C09504=6449,32951,-27517,288,-27969,-3249
C09505=6447,32929,-27544,288,-27961,-3248
C09506=6439,32909,-27568,289,-27953,-3245
C09507=6438,32887,-27595,290,-27945,-3245
C09508=6431,32867,-27619,291,-27937,-3242
C09509=6424,32847,-27644,292,-27930,-3239
C09510=6417,32826,-27669,293,-27922,-3237
C09511=6410,32806,-27694,294,-27914,-3234
C09512=6403,32785,-27719,295,-27907,-3231
C09513=6396,32765,-27743,296,-27899,-3228
C09514=6388,32745,-27768,298,-27891,-3226
C09515=6381,32724,-27793,299,-27884,-3223
C09516=6374,32704,-27818,300,-27876,-3220
C09517=6356,32692,-27833,302,-27871,-3213
C09518=6356,32692,-26433,302,-27871,-3213
C09519=5833,33315,-23080,374,-28099,-3008
C09520=5833,33315,-27080,374,-28099,-3008
C09521=5810,33311,-27085,378,-28097,-2999
C09522=5793,33299,-27099,380,-28093,-2992
C09523=5770,33296,-27104,384,-28091,-2983
C09524=5747,33292,-27108,387,-28090,-2974
C09525=5724,33289,-27112,390,-28088,-2965
C09526=5701,33286,-27117,393,-28087,-2956
C09527=5678,33282,-27121,397,-28085,-2947
C09528=5657,33289,-27113,400,-28087,-2939
C09529=5634,33286,-27117,403,-28086,-2930
C09530=5614,33292,-27109,406,-28088,-2922
C09531=5592,33293,-27109,409,-28088,-2914
C09532=5571,33295,-27106,412,-28089,-2906
C09533=5550,33298,-27103,415,-28090,-2897
C09534=5528,33299,-27102,418,-28090,-2889
C09535=5508,33305,-27094,421,-28092,-2881
C09536=5487,33309,-27090,424,-28093,-2873
C09537=5464,33309,-27091,427,-28093,-2864
C09538=5444,33315,-27083,430,-28095,-2856
C09539=5424,33322,-27075,433,-28097,-2848
C09540=5405,33333,-27061,435,-28101,-2841
C09541=5387,33345,-27047,438,-28106,-2834
C09542=5367,33353,-27038,441,-28108,-2826
C09543=5356,33370,-27017,442,-28115,-2821
C09544=5365,33371,-27016,441,-28115,-2825
C09545=5386,33365,-27023,438,-28113,-2833
C09546=5404,33351,-27039,435,-28108,-2840
C09547=5424,33345,-27046,433,-28106,-2848
C09548=5443,33334,-27060,430,-28102,-2856
C09549=5463,33328,-27068,427,-28100,-2864
C09550=5485,33327,-27068,424,-28100,-2872
C09551=5507,33324,-27071,421,-28099,-2880
C09552=5527,33318,-27079,418,-28097,-2888
C09553=5548,33316,-27081,415,-28096,-2897
C09554=5570,33314,-27083,412,-28096,-2905
C09555=5590,33308,-27091,409,-28094,-2913
C09556=5613,33311,-27086,406,-28095,-2922
C09557=5633,33305,-27094,403,-28093,-2930
C09558=5656,33308,-27090,400,-28095,-2939
C09559=5677,33301,-27098,397,-28092,-2947
C09560=5700,33305,-27094,394,-28094,-2956
C09561=5723,33308,-27089,390,-28095,-2965
C09562=5746,33311,-27085,387,-28097,-2974
C09563=5769,33315,-27081,384,-28098,-2982
C09564=5792,33318,-27076,380,-28100,-2991
C09565=5810,33329,-27063,378,-28104,-2999
C09566=5832,33334,-27056,375,-28106,-3007
C09567=5850,33346,-27042,372,-28111,-3014
C09568=5864,33364,-27020,370,-28118,-3019
C09569=5880,33379,-27002,367,-28124,-3026
C09570=5893,33394,-26983,366,-28129,-3031
C09571=5902,33413,-26960,364,-28137,-3034
C09572=5916,33431,-26938,362,-28144,-3040
C09573=5937,33427,-26943,359,-28142,-3048
C09574=5926,33410,-26964,361,-28136,-3043
C09575=5911,33392,-26986,363,-28129,-3038
C09576=5897,33374,-27008,365,-28122,-3033
C09577=5883,33356,-27030,367,-28115,-3027
C09578=5869,33339,-27051,369,-28108,-3021
C09579=5851,33327,-27065,372,-28104,-3015
C09580=5833,33315,-27080,374,-28099,-3008
C09581=5833,33315,-25680,374,-28099,-3008
C09582=5638,33727,-22582,400,-28251,-2930
C09583=5638,33727,-26582,400,-28251,-2930
C09584=5614,33723,-26586,404,-28250,-2921
C09585=5590,33720,-26591,407,-28248,-2911
C09586=5566,33716,-26595,410,-28246,-2902
C09587=5542,33713,-26600,414,-28245,-2893
C09588=5518,33709,-26604,417,-28243,-2883
C09589=5494,33706,-26609,421,-28242,-2874
C09590=5470,33702,-26613,424,-28240,-2865
C09591=5446,33699,-26618,427,-28238,-2855
C09592=5422,33695,-26622,431,-28237,-2846
C09593=5435,33707,-26608,429,-28241,-2851
C09594=5459,33710,-26604,426,-28243,-2860
C09595=5483,33714,-26599,422,-28244,-2870
C09596=5507,33717,-26595,419,-28246,-2879
C09597=5531,33721,-26590,415,-28248,-2888
C09598=5555,33724,-26586,412,-28249,-2898
C09599=5573,33736,-26571,409,-28254,-2905
C09600=5597,33740,-26566,406,-28256,-2914
C09601=5621,33743,-26562,402,-28257,-2924
C09602=5645,33747,-26557,399,-28259,-2933
C09603=5667,33754,-26549,396,-28262,-2941
C09604=5688,33763,-26538,393,-28265,-2949
C09605=5712,33766,-26533,389,-28267,-2959
C09606=5730,33779,-26518,387,-28272,-2966
C09607=5754,33782,-26514,383,-28273,-2975
C09608=5774,33792,-26502,380,-28277,-2983
C09609=5797,33798,-26494,377,-28280,-2992
C09610=5815,33810,-26479,374,-28284,-2999
C09611=5837,33817,-26471,371,-28287,-3008
C09612=5856,33830,-26455,369,-28292,-3015
C09613=5874,33842,-26440,366,-28297,-3022
C09614=5892,33855,-26424,363,-28302,-3029
C09615=5908,33872,-26404,361,-28308,-3035
C09616=5925,33886,-26386,358,-28314,-3042
C09617=5940,33905,-26363,356,-28321,-3047
C09618=5958,33917,-26348,354,-28326,-3055
C09619=5973,33936,-26325,352,-28333,-3060
C09620=5988,33955,-26302,349,-28340,-3066
C09621=6000,33974,-26279,347,-28348,-3071
C09622=6015,33978,-26273,345,-28350,-3076
C09623=6017,33959,-24896,345,-28342,-3077
C09624=-41004,59868,4099,4900,-34257,16705
C09625=-41004,59868,1099,4900,-34257,16705
C09626=-41004,64596,1380,5213,-31659,16463
C09627=-41004,59868,1099,4900,-34257,16705
C09628=-41004,59868,9099,4900,-34257,16705
C09629=6017,33959,-22296,345,-28342,-3077
C09630=6017,33959,-26296,345,-28342,-3077
C09631=6002,33941,-26319,347,-28335,-3072
C09632=5988,33922,-26342,349,-28328,-3066
C09633=5973,33903,-26365,352,-28321,-3060
C09634=5955,33891,-26380,354,-28316,-3053
C09635=5940,33872,-26403,356,-28309,-3048
C09636=5922,33859,-26419,359,-28304,-3041
C09637=5906,33843,-26439,361,-28298,-3034
C09638=5887,33830,-26454,364,-28293,-3027
C09639=5869,33818,-26469,367,-28288,-3020
C09640=5850,33806,-26484,370,-28283,-3013
C09641=5832,33793,-26499,372,-28278,-3006
C09642=5811,33784,-26511,375,-28274,-2998
C09643=5789,33778,-26519,378,-28272,-2989
C09644=5771,33765,-26534,381,-28267,-2982
C09645=5747,33762,-26538,384,-28265,-2972
C09646=5726,33752,-26550,387,-28262,-2965
C09647=5704,33746,-26558,391,-28259,-2956
C09648=5680,33743,-26562,394,-28257,-2947
C09649=5660,33733,-26573,397,-28254,-2939
C09650=5638,33727,-26582,400,-28251,-2930
C09651=5638,33727,-25182,400,-28251,-2930
C09652=5388,35827,-20036,425,-29034,-2826
C09653=5388,35827,-24036,425,-29034,-2826
C09654=5365,35833,-24029,428,-29036,-2816
C09655=5342,35839,-24021,431,-29038,-2807
C09656=5318,35845,-24014,434,-29040,-2798
C09657=5295,35851,-24007,438,-29042,-2789
C09658=5271,35857,-24000,441,-29044,-2780
C09659=5248,35863,-23993,444,-29046,-2770
C09660=5223,35866,-23990,448,-29047,-2761
C09661=5200,35874,-23980,451,-29050,-2752
C09662=5176,35876,-23979,454,-29050,-2742
C09663=5151,35878,-23976,457,-29050,-2732
C09664=5128,35884,-23969,461,-29052,-2723
C09665=5104,35887,-23965,464,-29053,-2714
C09666=5078,35886,-23967,468,-29052,-2704
C09667=5054,35890,-23962,471,-29054,-2694
C09668=5029,35888,-23965,474,-29053,-2684
C09669=5005,35893,-23959,478,-29054,-2675
C09670=4979,35891,-23963,481,-29053,-2665
C09671=4953,35887,-23968,485,-29051,-2655
C09672=4930,35893,-23960,488,-29053,-2645
C09673=4904,35889,-23965,492,-29051,-2635
C09674=4878,35885,-23970,495,-29049,-2625
C09675=4852,35881,-23975,499,-29047,-2615
C09676=4826,35877,-23980,503,-29046,-2604
C09677=4799,35874,-23985,506,-29044,-2594
C09678=4773,35870,-23990,510,-29042,-2584
C09679=4747,35866,-23995,513,-29040,-2574
C09680=4721,35862,-24000,517,-29038,-2564
C09681=4700,35849,-24016,520,-29033,-2555
C09682=4674,35845,-24021,524,-29032,-2545
C09683=4686,35862,-24001,522,-29038,-2550
C09684=4710,35870,-23991,519,-29041,-2559
C09685=4736,35874,-23986,515,-29043,-2569
C09686=4762,35878,-23981,511,-29045,-2579
C09687=4788,35881,-23976,508,-29047,-2590
C09688=4814,35885,-23971,504,-29048,-2600
C09689=4840,35889,-23966,500,-29050,-2610
C09690=4866,35893,-23961,497,-29052,-2620
C09691=4892,35897,-23956,493,-29054,-2631
C09692=4918,35901,-23951,490,-29056,-2641
C09693=4944,35905,-23946,486,-29057,-2651
C09694=4970,35908,-23941,482,-29059,-2661
C09695=4996,35912,-23936,479,-29061,-2671
C09696=5020,35906,-23943,476,-29059,-2681
C09697=5046,35910,-23938,472,-29061,-2691
C09698=5069,35904,-23945,469,-29059,-2700
C09699=5094,35903,-23946,465,-29059,-2710
C09700=5119,35902,-23948,462,-29059,-2720
C09701=5143,35900,-23950,458,-29058,-2729
C09702=5168,35898,-23951,455,-29058,-2739
C09703=5192,35893,-23957,452,-29057,-2748
C09704=5215,35887,-23964,449,-29055,-2757
C09705=5238,35881,-23971,445,-29053,-2767
C09706=5262,35875,-23978,442,-29051,-2776
C09707=5286,35870,-23985,439,-29049,-2785
C09708=5310,35868,-23986,435,-29049,-2795
C09709=5333,35860,-23996,432,-29046,-2804
C09710=5358,35858,-23998,429,-29046,-2814
C09711=5381,35849,-24008,426,-29043,-2823
C09712=5402,35834,-24027,423,-29037,-2831
C09713=5388,35827,-24036,425,-29034,-2826
C09714=5388,35827,-22636,425,-29034,-2826
C09715=5324,36018,-19804,433,-29105,-2800
C09716=5324,36018,-23804,433,-29105,-2800
C09717=5298,36029,-23791,436,-29109,-2790
C09718=5273,36040,-23779,440,-29112,-2780
C09719=5249,36057,-23757,443,-29119,-2770
C09720=5224,36068,-23745,446,-29122,-2760
C09721=5200,36085,-23724,450,-29129,-2751
C09722=5175,36096,-23711,453,-29132,-2741
C09723=5149,36107,-23699,457,-29136,-2731
C09724=5126,36123,-23679,460,-29142,-2721
C09725=5100,36135,-23665,463,-29146,-2712
C09726=5075,36144,-23654,467,-29149,-2701
C09727=5048,36150,-23647,470,-29151,-2691
C09728=5024,36166,-23629,474,-29156,-2681
C09729=4997,36171,-23622,477,-29158,-2671
C09730=4972,36181,-23611,481,-29161,-2661
C09731=4947,36191,-23598,484,-29165,-2651
C09732=4920,36198,-23590,488,-29167,-2640
C09733=4893,36204,-23584,491,-29169,-2630
C09734=4867,36209,-23577,495,-29170,-2620
C09735=4840,36215,-23571,499,-29172,-2609
C09736=4814,36223,-23561,502,-29175,-2599
C09737=4787,36227,-23557,506,-29176,-2588
C09738=4760,36232,-23551,510,-29177,-2578
C09739=4734,36237,-23545,513,-29179,-2567
C09740=4706,36238,-23545,517,-29179,-2556
C09741=4678,36239,-23544,521,-29179,-2545
C09742=4651,36244,-23537,524,-29180,-2535
C09743=4623,36241,-23541,528,-29179,-2523
C09744=4596,36246,-23536,532,-29180,-2513
C09745=4566,36241,-23542,536,-29178,-2501
C09746=4562,36258,-23522,537,-29184,-2500
C09747=4588,36254,-23526,533,-29183,-2510
C09748=4617,36258,-23521,529,-29185,-2521
C09749=4646,36263,-23515,525,-29187,-2533
C09750=4673,36257,-23522,521,-29185,-2543
C09751=4699,36252,-23528,518,-29184,-2554
C09752=4728,36255,-23524,514,-29185,-2565
C09753=4755,36250,-23529,510,-29184,-2575
C09754=4782,36245,-23535,507,-29182,-2586
C09755=4808,36239,-23542,503,-29181,-2596
C09756=4835,36233,-23549,499,-29179,-2607
C09757=4862,36230,-23553,496,-29178,-2618
C09758=4888,36222,-23562,492,-29175,-2628
C09759=4915,36216,-23568,488,-29174,-2638
C09760=4942,36211,-23575,485,-29172,-2649
C09761=4967,36201,-23586,481,-29169,-2659
C09762=4992,36191,-23598,478,-29165,-2669
C09763=5019,36184,-23606,474,-29163,-2679
C09764=5045,36177,-23615,471,-29161,-2690
C09765=5070,36163,-23631,467,-29156,-2699
C09766=5096,36155,-23640,464,-29153,-2710
C09767=5120,36141,-23657,460,-29149,-2719
C09768=5145,36127,-23674,457,-29143,-2729
C09769=5170,36116,-23686,454,-29140,-2739
C09770=5195,36106,-23699,450,-29136,-2749
C09771=5219,36089,-23719,447,-29130,-2758
C09772=5244,36078,-23733,444,-29126,-2768
C09773=5268,36060,-23754,440,-29120,-2778
C09774=5293,36049,-23766,437,-29116,-2788
C09775=5317,36032,-23788,434,-29110,-2797
C09776=5324,36018,-23804,433,-29105,-2800
C09777=5324,36018,-22404,433,-29105,-2800
C09778=5373,36428,-19306,424,-29259,-2818
C09779=5373,36428,-23306,424,-29259,-2818
C09780=5363,36436,-23296,426,-29262,-2814
C09781=5350,36436,-23296,427,-29262,-2809
C09782=5340,36444,-23287,429,-29265,-2805
C09783=5330,36452,-23277,430,-29268,-2801
C09784=5320,36460,-23268,431,-29271,-2797
C09785=5309,36467,-23259,433,-29273,-2793
C09786=5299,36475,-23250,434,-29276,-2789
C09787=5289,36483,-23240,436,-29279,-2785
C09788=5278,36491,-23231,437,-29282,-2780
C09789=5268,36498,-23222,438,-29284,-2776
C09790=5258,36506,-23213,440,-29287,-2772
C09791=5248,36514,-23203,441,-29290,-2768
C09792=5237,36521,-23194,442,-29293,-2764
C09793=5227,36529,-23185,444,-29295,-2760
C09794=5215,36530,-23184,446,-29295,-2755
C09795=5205,36538,-23175,447,-29298,-2751
C09796=5195,36545,-23166,448,-29301,-2747
C09797=5184,36553,-23156,450,-29304,-2743
C09798=5174,36561,-23147,451,-29306,-2739
C09799=5162,36561,-21746,453,-29306,-2734
C09800=-41004,59868,4099,4900,-34257,16705
C09801=-41004,59868,1099,4900,-34257,16705
C09802=-41004,64596,1380,5213,-31659,16463
C09803=-41004,59868,1099,4900,-34257,16705
C09804=-41004,59868,9099,4900,-34257,16705
C09805=5162,36561,-19146,453,-29306,-2734
C09806=5162,36561,-23146,453,-29306,-2734
C09807=5152,36569,-23137,454,-29309,-2730
C09808=5142,36577,-23128,455,-29312,-2726
C09809=5131,36584,-23120,457,-29314,-2722
C09810=5119,36585,-23118,458,-29315,-2718
C09811=5109,36593,-23109,460,-29317,-2713
C09812=5098,36598,-23103,461,-29319,-2709
C09813=5087,36601,-23099,463,-29320,-2705
C09814=5081,36612,-23086,464,-29324,-2702
C09815=5079,36624,-23072,464,-29329,-2702
C09816=5090,36616,-23081,462,-29326,-2706
C09817=5102,36615,-23082,461,-29326,-2711
C09818=5113,36610,-23088,459,-29324,-2715
C09819=5124,36607,-23092,458,-29323,-2719
C09820=5134,36599,-23101,456,-29320,-2723
C09821=5145,36592,-23110,455,-29317,-2727
C09822=5156,36588,-23115,453,-29316,-2732
C09823=5167,36583,-23120,452,-29315,-2736
C09824=5177,36575,-23129,451,-29312,-2740
C09825=5187,36568,-23139,449,-29309,-2744
C09826=5199,36565,-23141,448,-29308,-2749
C09827=5210,36559,-23148,446,-29306,-2753
C09828=5220,36552,-23158,445,-29304,-2757
C09829=5230,36544,-23167,443,-29301,-2761
C09830=5240,36536,-23176,442,-29298,-2765
C09831=5251,36528,-23186,441,-29295,-2769
C09832=5261,36521,-23195,439,-29293,-2773
C09833=5271,36513,-23204,438,-29290,-2778
C09834=5281,36505,-23213,437,-29287,-2782
C09835=5293,36502,-23216,435,-29286,-2786
C09836=5304,36497,-23223,433,-29284,-2790
C09837=5314,36489,-23232,432,-29281,-2794
C09838=5324,36481,-23242,431,-29279,-2799
C09839=5335,36474,-23251,429,-29276,-2803
C09840=5345,36466,-23260,428,-29273,-2807
C09841=5355,36458,-23269,427,-29271,-2811
C09842=5365,36450,-23279,425,-29268,-2815
C09843=5376,36443,-23288,424,-29265,-2819
C09844=5386,36435,-23297,422,-29262,-2823
C09845=5386,36430,-23303,423,-29260,-2823
C09846=5373,36428,-23306,424,-29259,-2818
C09847=5373,36428,-21906,424,-29259,-2818
//INST
///DATE 2026/04/29 10:00
///ATTR SC,RW
///GROUP1 RB1
NOP
MOVJ C00000 VJ=0.78
MOVJ C00001 VJ=0.78
MOVL C00002 V=11.7
TIMER T=2.00
MOVL C00003 V=11.7
MOVJ C00004 VJ=0.78
MOVJ C00005 VJ=0.78
MOVJ C00006 VJ=0.78
MOVL C00007 V=8.0
MOVL C00008 V=8.0
MOVL C00009 V=8.0
MOVL C00010 V=8.0
MOVL C00011 V=8.0
MOVL C00012 V=8.0
MOVL C00013 V=8.0
MOVL C00014 V=8.0
MOVL C00015 V=8.0
MOVL C00016 V=8.0
MOVL C00017 V=8.0
MOVL C00018 V=8.0
MOVL C00019 V=8.0
MOVL C00020 V=8.0
MOVL C00021 V=8.0
MOVL C00022 V=8.0
MOVL C00023 V=8.0
MOVL C00024 V=8.0
MOVL C00025 V=8.0
MOVL C00026 V=8.0
MOVL C00027 V=8.0
MOVL C00028 V=8.0
MOVL C00029 V=8.0
MOVL C00030 V=8.0
MOVL C00031 V=8.0
MOVL C00032 V=8.0
MOVL C00033 V=8.0
MOVL C00034 V=8.0
MOVL C00035 V=8.0
MOVL C00036 V=8.0
MOVL C00037 V=8.0
MOVL C00038 V=8.0
MOVL C00039 V=8.0
MOVL C00040 V=8.0
MOVL C00041 V=8.0
MOVL C00042 V=8.0
MOVL C00043 V=8.0
MOVL C00044 V=8.0
MOVL C00045 V=8.0
MOVL C00046 V=8.0
MOVL C00047 V=8.0
MOVL C00048 V=8.0
MOVL C00049 V=8.0
MOVL C00050 V=8.0
MOVL C00051 V=8.0
MOVL C00052 V=8.0
MOVL C00053 V=8.0
MOVL C00054 V=8.0
MOVL C00055 V=8.0
MOVL C00056 V=8.0
MOVL C00057 V=8.0
MOVL C00058 V=8.0
MOVL C00059 V=8.0
MOVL C00060 V=8.0
MOVL C00061 V=8.0
MOVL C00062 V=8.0
MOVL C00063 V=8.0
MOVL C00064 V=8.0
MOVL C00065 V=8.0
MOVL C00066 V=8.0
MOVL C00067 V=8.0
MOVL C00068 V=8.0
MOVJ C00069 VJ=0.78
MOVL C00070 V=8.0
MOVL C00071 V=8.0
MOVL C00072 V=8.0
MOVL C00073 V=8.0
MOVL C00074 V=8.0
MOVL C00075 V=8.0
MOVL C00076 V=8.0
MOVL C00077 V=8.0
MOVL C00078 V=8.0
MOVL C00079 V=8.0
MOVL C00080 V=8.0
MOVL C00081 V=8.0
MOVL C00082 V=8.0
MOVL C00083 V=8.0
MOVL C00084 V=8.0
MOVL C00085 V=8.0
MOVL C00086 V=8.0
MOVL C00087 V=8.0
MOVL C00088 V=8.0
MOVL C00089 V=8.0
MOVL C00090 V=8.0
MOVL C00091 V=8.0
MOVL C00092 V=8.0
MOVL C00093 V=8.0
MOVL C00094 V=8.0
MOVL C00095 V=8.0
MOVL C00096 V=8.0
MOVL C00097 V=8.0
MOVL C00098 V=8.0
MOVL C00099 V=8.0
MOVL C00100 V=8.0
MOVL C00101 V=8.0
MOVL C00102 V=8.0
MOVL C00103 V=8.0
MOVL C00104 V=8.0
MOVL C00105 V=8.0
MOVL C00106 V=8.0
MOVL C00107 V=8.0
MOVL C00108 V=8.0
MOVL C00109 V=8.0
MOVL C00110 V=8.0
MOVL C00111 V=8.0
MOVL C00112 V=8.0
MOVL C00113 V=8.0
MOVL C00114 V=8.0
MOVL C00115 V=8.0
MOVL C00116 V=8.0
MOVL C00117 V=8.0
MOVL C00118 V=8.0
MOVL C00119 V=8.0
MOVL C00120 V=8.0
MOVL C00121 V=8.0
MOVL C00122 V=8.0
MOVL C00123 V=8.0
MOVL C00124 V=8.0
MOVL C00125 V=8.0
MOVL C00126 V=8.0
MOVL C00127 V=8.0
MOVL C00128 V=8.0
MOVL C00129 V=8.0
MOVL C00130 V=8.0
MOVL C00131 V=8.0
MOVJ C00132 VJ=0.78
MOVL C00133 V=8.0
MOVL C00134 V=8.0
MOVL C00135 V=8.0
MOVL C00136 V=8.0
MOVL C00137 V=8.0
MOVL C00138 V=8.0
MOVL C00139 V=8.0
MOVL C00140 V=8.0
MOVL C00141 V=8.0
MOVL C00142 V=8.0
MOVL C00143 V=8.0
MOVL C00144 V=8.0
MOVL C00145 V=8.0
MOVL C00146 V=8.0
MOVL C00147 V=8.0
MOVL C00148 V=8.0
MOVL C00149 V=8.0
MOVL C00150 V=8.0
MOVL C00151 V=8.0
MOVL C00152 V=8.0
MOVL C00153 V=8.0
MOVL C00154 V=8.0
MOVL C00155 V=8.0
MOVL C00156 V=8.0
MOVL C00157 V=8.0
MOVL C00158 V=8.0
MOVL C00159 V=8.0
MOVL C00160 V=8.0
MOVL C00161 V=8.0
MOVL C00162 V=8.0
MOVL C00163 V=8.0
MOVL C00164 V=8.0
MOVL C00165 V=8.0
MOVL C00166 V=8.0
MOVL C00167 V=8.0
MOVL C00168 V=8.0
MOVL C00169 V=8.0
MOVL C00170 V=8.0
MOVL C00171 V=8.0
MOVL C00172 V=8.0
MOVL C00173 V=8.0
MOVJ C00174 VJ=0.78
MOVJ C00175 VJ=0.78
MOVL C00176 V=11.7
TIMER T=2.00
MOVL C00177 V=11.7
MOVJ C00178 VJ=0.78
MOVJ C00179 VJ=0.78
MOVL C00180 V=8.0
MOVL C00181 V=8.0
MOVL C00182 V=8.0
MOVL C00183 V=8.0
MOVL C00184 V=8.0
MOVL C00185 V=8.0
MOVL C00186 V=8.0
MOVL C00187 V=8.0
MOVL C00188 V=8.0
MOVL C00189 V=8.0
MOVL C00190 V=8.0
MOVL C00191 V=8.0
MOVL C00192 V=8.0
MOVL C00193 V=8.0
MOVL C00194 V=8.0
MOVL C00195 V=8.0
MOVL C00196 V=8.0
MOVL C00197 V=8.0
MOVL C00198 V=8.0
MOVL C00199 V=8.0
MOVL C00200 V=8.0
MOVL C00201 V=8.0
MOVJ C00202 VJ=0.78
MOVL C00203 V=8.0
MOVL C00204 V=8.0
MOVL C00205 V=8.0
MOVL C00206 V=8.0
MOVL C00207 V=8.0
MOVL C00208 V=8.0
MOVL C00209 V=8.0
MOVL C00210 V=8.0
MOVL C00211 V=8.0
MOVL C00212 V=8.0
MOVL C00213 V=8.0
MOVL C00214 V=8.0
MOVL C00215 V=8.0
MOVL C00216 V=8.0
MOVL C00217 V=8.0
MOVL C00218 V=8.0
MOVL C00219 V=8.0
MOVL C00220 V=8.0
MOVL C00221 V=8.0
MOVL C00222 V=8.0
MOVL C00223 V=8.0
MOVL C00224 V=8.0
MOVL C00225 V=8.0
MOVL C00226 V=8.0
MOVL C00227 V=8.0
MOVL C00228 V=8.0
MOVL C00229 V=8.0
MOVL C00230 V=8.0
MOVL C00231 V=8.0
MOVL C00232 V=8.0
MOVL C00233 V=8.0
MOVL C00234 V=8.0
MOVL C00235 V=8.0
MOVL C00236 V=8.0
MOVL C00237 V=8.0
MOVL C00238 V=8.0
MOVL C00239 V=8.0
MOVL C00240 V=8.0
MOVL C00241 V=8.0
MOVL C00242 V=8.0
MOVL C00243 V=8.0
MOVL C00244 V=8.0
MOVL C00245 V=8.0
MOVL C00246 V=8.0
MOVL C00247 V=8.0
MOVL C00248 V=8.0
MOVL C00249 V=8.0
MOVL C00250 V=8.0
MOVL C00251 V=8.0
MOVL C00252 V=8.0
MOVL C00253 V=8.0
MOVL C00254 V=8.0
MOVL C00255 V=8.0
MOVL C00256 V=8.0
MOVL C00257 V=8.0
MOVL C00258 V=8.0
MOVL C00259 V=8.0
MOVL C00260 V=8.0
MOVL C00261 V=8.0
MOVL C00262 V=8.0
MOVL C00263 V=8.0
MOVL C00264 V=8.0
MOVJ C00265 VJ=0.78
MOVL C00266 V=8.0
MOVL C00267 V=8.0
MOVL C00268 V=8.0
MOVL C00269 V=8.0
MOVL C00270 V=8.0
MOVL C00271 V=8.0
MOVL C00272 V=8.0
MOVL C00273 V=8.0
MOVL C00274 V=8.0
MOVL C00275 V=8.0
MOVL C00276 V=8.0
MOVL C00277 V=8.0
MOVL C00278 V=8.0
MOVL C00279 V=8.0
MOVL C00280 V=8.0
MOVL C00281 V=8.0
MOVL C00282 V=8.0
MOVL C00283 V=8.0
MOVL C00284 V=8.0
MOVL C00285 V=8.0
MOVL C00286 V=8.0
MOVL C00287 V=8.0
MOVL C00288 V=8.0
MOVL C00289 V=8.0
MOVL C00290 V=8.0
MOVL C00291 V=8.0
MOVL C00292 V=8.0
MOVL C00293 V=8.0
MOVL C00294 V=8.0
MOVL C00295 V=8.0
MOVL C00296 V=8.0
MOVL C00297 V=8.0
MOVL C00298 V=8.0
MOVL C00299 V=8.0
MOVL C00300 V=8.0
MOVL C00301 V=8.0
MOVL C00302 V=8.0
MOVL C00303 V=8.0
MOVL C00304 V=8.0
MOVL C00305 V=8.0
MOVL C00306 V=8.0
MOVL C00307 V=8.0
MOVL C00308 V=8.0
MOVL C00309 V=8.0
MOVL C00310 V=8.0
MOVL C00311 V=8.0
MOVL C00312 V=8.0
MOVL C00313 V=8.0
MOVL C00314 V=8.0
MOVL C00315 V=8.0
MOVL C00316 V=8.0
MOVL C00317 V=8.0
MOVL C00318 V=8.0
MOVL C00319 V=8.0
MOVL C00320 V=8.0
MOVL C00321 V=8.0
MOVL C00322 V=8.0
MOVL C00323 V=8.0
MOVL C00324 V=8.0
MOVL C00325 V=8.0
MOVL C00326 V=8.0
MOVL C00327 V=8.0
MOVJ C00328 VJ=0.78
MOVL C00329 V=8.0
MOVL C00330 V=8.0
MOVL C00331 V=8.0
MOVL C00332 V=8.0
MOVL C00333 V=8.0
MOVL C00334 V=8.0
MOVL C00335 V=8.0
MOVL C00336 V=8.0
MOVL C00337 V=8.0
MOVL C00338 V=8.0
MOVL C00339 V=8.0
MOVL C00340 V=8.0
MOVL C00341 V=8.0
MOVL C00342 V=8.0
MOVL C00343 V=8.0
MOVL C00344 V=8.0
MOVL C00345 V=8.0
MOVL C00346 V=8.0
MOVL C00347 V=8.0
MOVL C00348 V=8.0
MOVL C00349 V=8.0
MOVJ C00350 VJ=0.78
MOVJ C00351 VJ=0.78
MOVL C00352 V=11.7
TIMER T=2.00
MOVL C00353 V=11.7
MOVJ C00354 VJ=0.78
MOVJ C00355 VJ=0.78
MOVL C00356 V=8.0
MOVL C00357 V=8.0
MOVL C00358 V=8.0
MOVL C00359 V=8.0
MOVL C00360 V=8.0
MOVL C00361 V=8.0
MOVL C00362 V=8.0
MOVL C00363 V=8.0
MOVL C00364 V=8.0
MOVL C00365 V=8.0
MOVL C00366 V=8.0
MOVL C00367 V=8.0
MOVL C00368 V=8.0
MOVL C00369 V=8.0
MOVL C00370 V=8.0
MOVL C00371 V=8.0
MOVL C00372 V=8.0
MOVL C00373 V=8.0
MOVL C00374 V=8.0
MOVL C00375 V=8.0
MOVL C00376 V=8.0
MOVL C00377 V=8.0
MOVL C00378 V=8.0
MOVL C00379 V=8.0
MOVL C00380 V=8.0
MOVL C00381 V=8.0
MOVL C00382 V=8.0
MOVL C00383 V=8.0
MOVL C00384 V=8.0
MOVL C00385 V=8.0
MOVL C00386 V=8.0
MOVL C00387 V=8.0
MOVL C00388 V=8.0
MOVL C00389 V=8.0
MOVL C00390 V=8.0
MOVL C00391 V=8.0
MOVL C00392 V=8.0
MOVL C00393 V=8.0
MOVL C00394 V=8.0
MOVL C00395 V=8.0
MOVL C00396 V=8.0
MOVL C00397 V=8.0
MOVJ C00398 VJ=0.78
MOVL C00399 V=8.0
MOVL C00400 V=8.0
MOVL C00401 V=8.0
MOVL C00402 V=8.0
MOVL C00403 V=8.0
MOVL C00404 V=8.0
MOVL C00405 V=8.0
MOVL C00406 V=8.0
MOVL C00407 V=8.0
MOVL C00408 V=8.0
MOVL C00409 V=8.0
MOVL C00410 V=8.0
MOVL C00411 V=8.0
MOVL C00412 V=8.0
MOVL C00413 V=8.0
MOVL C00414 V=8.0
MOVL C00415 V=8.0
MOVL C00416 V=8.0
MOVL C00417 V=8.0
MOVL C00418 V=8.0
MOVL C00419 V=8.0
MOVL C00420 V=8.0
MOVL C00421 V=8.0
MOVL C00422 V=8.0
MOVL C00423 V=8.0
MOVL C00424 V=8.0
MOVL C00425 V=8.0
MOVL C00426 V=8.0
MOVL C00427 V=8.0
MOVL C00428 V=8.0
MOVL C00429 V=8.0
MOVL C00430 V=8.0
MOVL C00431 V=8.0
MOVL C00432 V=8.0
MOVL C00433 V=8.0
MOVL C00434 V=8.0
MOVL C00435 V=8.0
MOVL C00436 V=8.0
MOVL C00437 V=8.0
MOVL C00438 V=8.0
MOVL C00439 V=8.0
MOVL C00440 V=8.0
MOVL C00441 V=8.0
MOVL C00442 V=8.0
MOVL C00443 V=8.0
MOVL C00444 V=8.0
MOVL C00445 V=8.0
MOVL C00446 V=8.0
MOVL C00447 V=8.0
MOVL C00448 V=8.0
MOVL C00449 V=8.0
MOVL C00450 V=8.0
MOVL C00451 V=8.0
MOVL C00452 V=8.0
MOVL C00453 V=8.0
MOVL C00454 V=8.0
MOVL C00455 V=8.0
MOVL C00456 V=8.0
MOVL C00457 V=8.0
MOVL C00458 V=8.0
MOVL C00459 V=8.0
MOVL C00460 V=8.0
MOVJ C00461 VJ=0.78
MOVL C00462 V=8.0
MOVL C00463 V=8.0
MOVL C00464 V=8.0
MOVL C00465 V=8.0
MOVL C00466 V=8.0
MOVL C00467 V=8.0
MOVL C00468 V=8.0
MOVL C00469 V=8.0
MOVL C00470 V=8.0
MOVL C00471 V=8.0
MOVL C00472 V=8.0
MOVL C00473 V=8.0
MOVL C00474 V=8.0
MOVL C00475 V=8.0
MOVL C00476 V=8.0
MOVL C00477 V=8.0
MOVL C00478 V=8.0
MOVL C00479 V=8.0
MOVL C00480 V=8.0
MOVL C00481 V=8.0
MOVL C00482 V=8.0
MOVL C00483 V=8.0
MOVL C00484 V=8.0
MOVL C00485 V=8.0
MOVL C00486 V=8.0
MOVL C00487 V=8.0
MOVL C00488 V=8.0
MOVL C00489 V=8.0
MOVL C00490 V=8.0
MOVL C00491 V=8.0
MOVL C00492 V=8.0
MOVL C00493 V=8.0
MOVL C00494 V=8.0
MOVL C00495 V=8.0
MOVL C00496 V=8.0
MOVL C00497 V=8.0
MOVL C00498 V=8.0
MOVL C00499 V=8.0
MOVL C00500 V=8.0
MOVL C00501 V=8.0
MOVL C00502 V=8.0
MOVL C00503 V=8.0
MOVL C00504 V=8.0
MOVL C00505 V=8.0
MOVL C00506 V=8.0
MOVL C00507 V=8.0
MOVL C00508 V=8.0
MOVL C00509 V=8.0
MOVL C00510 V=8.0
MOVL C00511 V=8.0
MOVL C00512 V=8.0
MOVL C00513 V=8.0
MOVL C00514 V=8.0
MOVL C00515 V=8.0
MOVL C00516 V=8.0
MOVL C00517 V=8.0
MOVL C00518 V=8.0
MOVL C00519 V=8.0
MOVL C00520 V=8.0
MOVL C00521 V=8.0
MOVL C00522 V=8.0
MOVJ C00523 VJ=0.78
MOVJ C00524 VJ=0.78
MOVL C00525 V=11.7
TIMER T=2.00
MOVL C00526 V=11.7
MOVJ C00527 VJ=0.78
MOVJ C00528 VJ=0.78
MOVL C00529 V=8.0
MOVL C00530 V=8.0
MOVJ C00531 VJ=0.78
MOVL C00532 V=8.0
MOVL C00533 V=8.0
MOVL C00534 V=8.0
MOVL C00535 V=8.0
MOVL C00536 V=8.0
MOVL C00537 V=8.0
MOVL C00538 V=8.0
MOVL C00539 V=8.0
MOVL C00540 V=8.0
MOVL C00541 V=8.0
MOVL C00542 V=8.0
MOVL C00543 V=8.0
MOVL C00544 V=8.0
MOVL C00545 V=8.0
MOVL C00546 V=8.0
MOVL C00547 V=8.0
MOVL C00548 V=8.0
MOVL C00549 V=8.0
MOVL C00550 V=8.0
MOVL C00551 V=8.0
MOVL C00552 V=8.0
MOVL C00553 V=8.0
MOVL C00554 V=8.0
MOVL C00555 V=8.0
MOVL C00556 V=8.0
MOVL C00557 V=8.0
MOVL C00558 V=8.0
MOVL C00559 V=8.0
MOVL C00560 V=8.0
MOVL C00561 V=8.0
MOVL C00562 V=8.0
MOVL C00563 V=8.0
MOVL C00564 V=8.0
MOVL C00565 V=8.0
MOVL C00566 V=8.0
MOVL C00567 V=8.0
MOVL C00568 V=8.0
MOVL C00569 V=8.0
MOVL C00570 V=8.0
MOVL C00571 V=8.0
MOVL C00572 V=8.0
MOVL C00573 V=8.0
MOVL C00574 V=8.0
MOVL C00575 V=8.0
MOVL C00576 V=8.0
MOVL C00577 V=8.0
MOVL C00578 V=8.0
MOVL C00579 V=8.0
MOVL C00580 V=8.0
MOVL C00581 V=8.0
MOVL C00582 V=8.0
MOVL C00583 V=8.0
MOVL C00584 V=8.0
MOVL C00585 V=8.0
MOVL C00586 V=8.0
MOVL C00587 V=8.0
MOVL C00588 V=8.0
MOVL C00589 V=8.0
MOVL C00590 V=8.0
MOVL C00591 V=8.0
MOVL C00592 V=8.0
MOVL C00593 V=8.0
MOVJ C00594 VJ=0.78
MOVL C00595 V=8.0
MOVL C00596 V=8.0
MOVL C00597 V=8.0
MOVL C00598 V=8.0
MOVL C00599 V=8.0
MOVL C00600 V=8.0
MOVL C00601 V=8.0
MOVL C00602 V=8.0
MOVL C00603 V=8.0
MOVL C00604 V=8.0
MOVL C00605 V=8.0
MOVL C00606 V=8.0
MOVL C00607 V=8.0
MOVL C00608 V=8.0
MOVL C00609 V=8.0
MOVL C00610 V=8.0
MOVL C00611 V=8.0
MOVL C00612 V=8.0
MOVL C00613 V=8.0
MOVL C00614 V=8.0
MOVL C00615 V=8.0
MOVL C00616 V=8.0
MOVL C00617 V=8.0
MOVL C00618 V=8.0
MOVL C00619 V=8.0
MOVL C00620 V=8.0
MOVL C00621 V=8.0
MOVL C00622 V=8.0
MOVL C00623 V=8.0
MOVL C00624 V=8.0
MOVL C00625 V=8.0
MOVL C00626 V=8.0
MOVL C00627 V=8.0
MOVL C00628 V=8.0
MOVL C00629 V=8.0
MOVL C00630 V=8.0
MOVL C00631 V=8.0
MOVL C00632 V=8.0
MOVL C00633 V=8.0
MOVL C00634 V=8.0
MOVL C00635 V=8.0
MOVL C00636 V=8.0
MOVL C00637 V=8.0
MOVL C00638 V=8.0
MOVL C00639 V=8.0
MOVL C00640 V=8.0
MOVL C00641 V=8.0
MOVL C00642 V=8.0
MOVL C00643 V=8.0
MOVL C00644 V=8.0
MOVL C00645 V=8.0
MOVL C00646 V=8.0
MOVL C00647 V=8.0
MOVL C00648 V=8.0
MOVL C00649 V=8.0
MOVL C00650 V=8.0
MOVL C00651 V=8.0
MOVL C00652 V=8.0
MOVL C00653 V=8.0
MOVL C00654 V=8.0
MOVL C00655 V=8.0
MOVL C00656 V=8.0
MOVJ C00657 VJ=0.78
MOVL C00658 V=8.0
MOVL C00659 V=8.0
MOVL C00660 V=8.0
MOVL C00661 V=8.0
MOVL C00662 V=8.0
MOVL C00663 V=8.0
MOVL C00664 V=8.0
MOVL C00665 V=8.0
MOVL C00666 V=8.0
MOVL C00667 V=8.0
MOVL C00668 V=8.0
MOVL C00669 V=8.0
MOVL C00670 V=8.0
MOVL C00671 V=8.0
MOVL C00672 V=8.0
MOVL C00673 V=8.0
MOVL C00674 V=8.0
MOVL C00675 V=8.0
MOVL C00676 V=8.0
MOVL C00677 V=8.0
MOVL C00678 V=8.0
MOVL C00679 V=8.0
MOVL C00680 V=8.0
MOVL C00681 V=8.0
MOVL C00682 V=8.0
MOVL C00683 V=8.0
MOVL C00684 V=8.0
MOVL C00685 V=8.0
MOVL C00686 V=8.0
MOVL C00687 V=8.0
MOVL C00688 V=8.0
MOVL C00689 V=8.0
MOVL C00690 V=8.0
MOVL C00691 V=8.0
MOVL C00692 V=8.0
MOVL C00693 V=8.0
MOVL C00694 V=8.0
MOVL C00695 V=8.0
MOVL C00696 V=8.0
MOVL C00697 V=8.0
MOVL C00698 V=8.0
MOVJ C00699 VJ=0.78
MOVJ C00700 VJ=0.78
MOVL C00701 V=11.7
TIMER T=2.00
MOVL C00702 V=11.7
MOVJ C00703 VJ=0.78
MOVJ C00704 VJ=0.78
MOVL C00705 V=8.0
MOVL C00706 V=8.0
MOVL C00707 V=8.0
MOVL C00708 V=8.0
MOVL C00709 V=8.0
MOVL C00710 V=8.0
MOVL C00711 V=8.0
MOVL C00712 V=8.0
MOVL C00713 V=8.0
MOVL C00714 V=8.0
MOVL C00715 V=8.0
MOVL C00716 V=8.0
MOVL C00717 V=8.0
MOVL C00718 V=8.0
MOVL C00719 V=8.0
MOVL C00720 V=8.0
MOVL C00721 V=8.0
MOVL C00722 V=8.0
MOVL C00723 V=8.0
MOVL C00724 V=8.0
MOVL C00725 V=8.0
MOVL C00726 V=8.0
MOVJ C00727 VJ=0.78
MOVL C00728 V=8.0
MOVL C00729 V=8.0
MOVL C00730 V=8.0
MOVL C00731 V=8.0
MOVL C00732 V=8.0
MOVL C00733 V=8.0
MOVL C00734 V=8.0
MOVL C00735 V=8.0
MOVL C00736 V=8.0
MOVL C00737 V=8.0
MOVL C00738 V=8.0
MOVL C00739 V=8.0
MOVL C00740 V=8.0
MOVL C00741 V=8.0
MOVL C00742 V=8.0
MOVL C00743 V=8.0
MOVL C00744 V=8.0
MOVL C00745 V=8.0
MOVL C00746 V=8.0
MOVL C00747 V=8.0
MOVL C00748 V=8.0
MOVL C00749 V=8.0
MOVL C00750 V=8.0
MOVL C00751 V=8.0
MOVL C00752 V=8.0
MOVL C00753 V=8.0
MOVL C00754 V=8.0
MOVL C00755 V=8.0
MOVL C00756 V=8.0
MOVL C00757 V=8.0
MOVL C00758 V=8.0
MOVL C00759 V=8.0
MOVL C00760 V=8.0
MOVL C00761 V=8.0
MOVL C00762 V=8.0
MOVL C00763 V=8.0
MOVL C00764 V=8.0
MOVL C00765 V=8.0
MOVL C00766 V=8.0
MOVL C00767 V=8.0
MOVL C00768 V=8.0
MOVL C00769 V=8.0
MOVL C00770 V=8.0
MOVL C00771 V=8.0
MOVL C00772 V=8.0
MOVL C00773 V=8.0
MOVL C00774 V=8.0
MOVL C00775 V=8.0
MOVL C00776 V=8.0
MOVL C00777 V=8.0
MOVL C00778 V=8.0
MOVL C00779 V=8.0
MOVL C00780 V=8.0
MOVL C00781 V=8.0
MOVL C00782 V=8.0
MOVL C00783 V=8.0
MOVL C00784 V=8.0
MOVL C00785 V=8.0
MOVL C00786 V=8.0
MOVL C00787 V=8.0
MOVL C00788 V=8.0
MOVL C00789 V=8.0
MOVJ C00790 VJ=0.78
MOVL C00791 V=8.0
MOVL C00792 V=8.0
MOVL C00793 V=8.0
MOVL C00794 V=8.0
MOVL C00795 V=8.0
MOVL C00796 V=8.0
MOVL C00797 V=8.0
MOVL C00798 V=8.0
MOVL C00799 V=8.0
MOVL C00800 V=8.0
MOVL C00801 V=8.0
MOVL C00802 V=8.0
MOVL C00803 V=8.0
MOVL C00804 V=8.0
MOVL C00805 V=8.0
MOVL C00806 V=8.0
MOVL C00807 V=8.0
MOVL C00808 V=8.0
MOVL C00809 V=8.0
MOVL C00810 V=8.0
MOVL C00811 V=8.0
MOVL C00812 V=8.0
MOVL C00813 V=8.0
MOVL C00814 V=8.0
MOVL C00815 V=8.0
MOVL C00816 V=8.0
MOVL C00817 V=8.0
MOVL C00818 V=8.0
MOVL C00819 V=8.0
MOVL C00820 V=8.0
MOVL C00821 V=8.0
MOVL C00822 V=8.0
MOVL C00823 V=8.0
MOVL C00824 V=8.0
MOVL C00825 V=8.0
MOVL C00826 V=8.0
MOVL C00827 V=8.0
MOVL C00828 V=8.0
MOVL C00829 V=8.0
MOVL C00830 V=8.0
MOVL C00831 V=8.0
MOVL C00832 V=8.0
MOVL C00833 V=8.0
MOVL C00834 V=8.0
MOVL C00835 V=8.0
MOVL C00836 V=8.0
MOVL C00837 V=8.0
MOVL C00838 V=8.0
MOVL C00839 V=8.0
MOVL C00840 V=8.0
MOVL C00841 V=8.0
MOVL C00842 V=8.0
MOVL C00843 V=8.0
MOVL C00844 V=8.0
MOVL C00845 V=8.0
MOVL C00846 V=8.0
MOVL C00847 V=8.0
MOVL C00848 V=8.0
MOVL C00849 V=8.0
MOVL C00850 V=8.0
MOVL C00851 V=8.0
MOVL C00852 V=8.0
MOVJ C00853 VJ=0.78
MOVL C00854 V=8.0
MOVL C00855 V=8.0
MOVL C00856 V=8.0
MOVL C00857 V=8.0
MOVL C00858 V=8.0
MOVL C00859 V=8.0
MOVL C00860 V=8.0
MOVL C00861 V=8.0
MOVL C00862 V=8.0
MOVL C00863 V=8.0
MOVL C00864 V=8.0
MOVL C00865 V=8.0
MOVL C00866 V=8.0
MOVL C00867 V=8.0
MOVL C00868 V=8.0
MOVL C00869 V=8.0
MOVL C00870 V=8.0
MOVL C00871 V=8.0
MOVL C00872 V=8.0
MOVL C00873 V=8.0
MOVL C00874 V=8.0
MOVJ C00875 VJ=0.78
MOVJ C00876 VJ=0.78
MOVL C00877 V=11.7
TIMER T=2.00
MOVL C00878 V=11.7
MOVJ C00879 VJ=0.78
MOVJ C00880 VJ=0.78
MOVL C00881 V=8.0
MOVL C00882 V=8.0
MOVL C00883 V=8.0
MOVL C00884 V=8.0
MOVL C00885 V=8.0
MOVL C00886 V=8.0
MOVL C00887 V=8.0
MOVL C00888 V=8.0
MOVL C00889 V=8.0
MOVL C00890 V=8.0
MOVL C00891 V=8.0
MOVL C00892 V=8.0
MOVL C00893 V=8.0
MOVL C00894 V=8.0
MOVL C00895 V=8.0
MOVL C00896 V=8.0
MOVL C00897 V=8.0
MOVL C00898 V=8.0
MOVL C00899 V=8.0
MOVL C00900 V=8.0
MOVL C00901 V=8.0
MOVL C00902 V=8.0
MOVL C00903 V=8.0
MOVL C00904 V=8.0
MOVL C00905 V=8.0
MOVL C00906 V=8.0
MOVL C00907 V=8.0
MOVL C00908 V=8.0
MOVL C00909 V=8.0
MOVL C00910 V=8.0
MOVL C00911 V=8.0
MOVL C00912 V=8.0
MOVL C00913 V=8.0
MOVL C00914 V=8.0
MOVL C00915 V=8.0
MOVL C00916 V=8.0
MOVL C00917 V=8.0
MOVL C00918 V=8.0
MOVL C00919 V=8.0
MOVL C00920 V=8.0
MOVL C00921 V=8.0
MOVL C00922 V=8.0
MOVJ C00923 VJ=0.78
MOVL C00924 V=8.0
MOVL C00925 V=8.0
MOVL C00926 V=8.0
MOVL C00927 V=8.0
MOVL C00928 V=8.0
MOVL C00929 V=8.0
MOVL C00930 V=8.0
MOVL C00931 V=8.0
MOVL C00932 V=8.0
MOVL C00933 V=8.0
MOVL C00934 V=8.0
MOVL C00935 V=8.0
MOVL C00936 V=8.0
MOVL C00937 V=8.0
MOVL C00938 V=8.0
MOVL C00939 V=8.0
MOVL C00940 V=8.0
MOVL C00941 V=8.0
MOVL C00942 V=8.0
MOVL C00943 V=8.0
MOVL C00944 V=8.0
MOVL C00945 V=8.0
MOVL C00946 V=8.0
MOVL C00947 V=8.0
MOVL C00948 V=8.0
MOVL C00949 V=8.0
MOVL C00950 V=8.0
MOVL C00951 V=8.0
MOVL C00952 V=8.0
MOVL C00953 V=8.0
MOVL C00954 V=8.0
MOVL C00955 V=8.0
MOVL C00956 V=8.0
MOVL C00957 V=8.0
MOVL C00958 V=8.0
MOVL C00959 V=8.0
MOVL C00960 V=8.0
MOVL C00961 V=8.0
MOVL C00962 V=8.0
MOVL C00963 V=8.0
MOVL C00964 V=8.0
MOVL C00965 V=8.0
MOVL C00966 V=8.0
MOVL C00967 V=8.0
MOVL C00968 V=8.0
MOVL C00969 V=8.0
MOVL C00970 V=8.0
MOVL C00971 V=8.0
MOVL C00972 V=8.0
MOVL C00973 V=8.0
MOVL C00974 V=8.0
MOVL C00975 V=8.0
MOVL C00976 V=8.0
MOVL C00977 V=8.0
MOVL C00978 V=8.0
MOVL C00979 V=8.0
MOVL C00980 V=8.0
MOVL C00981 V=8.0
MOVL C00982 V=8.0
MOVL C00983 V=8.0
MOVL C00984 V=8.0
MOVL C00985 V=8.0
MOVJ C00986 VJ=0.78
MOVL C00987 V=8.0
MOVL C00988 V=8.0
MOVL C00989 V=8.0
MOVL C00990 V=8.0
MOVL C00991 V=8.0
MOVL C00992 V=8.0
MOVL C00993 V=8.0
MOVL C00994 V=8.0
MOVL C00995 V=8.0
MOVL C00996 V=8.0
MOVL C00997 V=8.0
MOVL C00998 V=8.0
MOVL C00999 V=8.0
MOVL C01000 V=8.0
MOVL C01001 V=8.0
MOVL C01002 V=8.0
MOVL C01003 V=8.0
MOVL C01004 V=8.0
MOVL C01005 V=8.0
MOVL C01006 V=8.0
MOVL C01007 V=8.0
MOVL C01008 V=8.0
MOVL C01009 V=8.0
MOVL C01010 V=8.0
MOVL C01011 V=8.0
MOVL C01012 V=8.0
MOVL C01013 V=8.0
MOVL C01014 V=8.0
MOVL C01015 V=8.0
MOVL C01016 V=8.0
MOVL C01017 V=8.0
MOVL C01018 V=8.0
MOVL C01019 V=8.0
MOVL C01020 V=8.0
MOVL C01021 V=8.0
MOVL C01022 V=8.0
MOVL C01023 V=8.0
MOVL C01024 V=8.0
MOVL C01025 V=8.0
MOVL C01026 V=8.0
MOVL C01027 V=8.0
MOVL C01028 V=8.0
MOVL C01029 V=8.0
MOVL C01030 V=8.0
MOVL C01031 V=8.0
MOVL C01032 V=8.0
MOVL C01033 V=8.0
MOVL C01034 V=8.0
MOVL C01035 V=8.0
MOVL C01036 V=8.0
MOVL C01037 V=8.0
MOVL C01038 V=8.0
MOVL C01039 V=8.0
MOVL C01040 V=8.0
MOVL C01041 V=8.0
MOVL C01042 V=8.0
MOVL C01043 V=8.0
MOVL C01044 V=8.0
MOVL C01045 V=8.0
MOVL C01046 V=8.0
MOVL C01047 V=8.0
MOVJ C01048 VJ=0.78
MOVJ C01049 VJ=0.78
MOVL C01050 V=11.7
TIMER T=2.00
MOVL C01051 V=11.7
MOVJ C01052 VJ=0.78
MOVJ C01053 VJ=0.78
MOVL C01054 V=8.0
MOVL C01055 V=8.0
MOVJ C01056 VJ=0.78
MOVL C01057 V=8.0
MOVL C01058 V=8.0
MOVL C01059 V=8.0
MOVL C01060 V=8.0
MOVL C01061 V=8.0
MOVL C01062 V=8.0
MOVL C01063 V=8.0
MOVL C01064 V=8.0
MOVL C01065 V=8.0
MOVL C01066 V=8.0
MOVL C01067 V=8.0
MOVL C01068 V=8.0
MOVL C01069 V=8.0
MOVL C01070 V=8.0
MOVL C01071 V=8.0
MOVL C01072 V=8.0
MOVL C01073 V=8.0
MOVL C01074 V=8.0
MOVL C01075 V=8.0
MOVL C01076 V=8.0
MOVL C01077 V=8.0
MOVL C01078 V=8.0
MOVL C01079 V=8.0
MOVL C01080 V=8.0
MOVL C01081 V=8.0
MOVL C01082 V=8.0
MOVL C01083 V=8.0
MOVL C01084 V=8.0
MOVL C01085 V=8.0
MOVL C01086 V=8.0
MOVL C01087 V=8.0
MOVL C01088 V=8.0
MOVL C01089 V=8.0
MOVL C01090 V=8.0
MOVL C01091 V=8.0
MOVL C01092 V=8.0
MOVL C01093 V=8.0
MOVL C01094 V=8.0
MOVL C01095 V=8.0
MOVL C01096 V=8.0
MOVL C01097 V=8.0
MOVL C01098 V=8.0
MOVL C01099 V=8.0
MOVL C01100 V=8.0
MOVL C01101 V=8.0
MOVL C01102 V=8.0
MOVL C01103 V=8.0
MOVL C01104 V=8.0
MOVL C01105 V=8.0
MOVL C01106 V=8.0
MOVL C01107 V=8.0
MOVL C01108 V=8.0
MOVL C01109 V=8.0
MOVL C01110 V=8.0
MOVL C01111 V=8.0
MOVL C01112 V=8.0
MOVL C01113 V=8.0
MOVL C01114 V=8.0
MOVL C01115 V=8.0
MOVL C01116 V=8.0
MOVL C01117 V=8.0
MOVL C01118 V=8.0
MOVJ C01119 VJ=0.78
MOVL C01120 V=8.0
MOVL C01121 V=8.0
MOVL C01122 V=8.0
MOVL C01123 V=8.0
MOVL C01124 V=8.0
MOVL C01125 V=8.0
MOVL C01126 V=8.0
MOVL C01127 V=8.0
MOVL C01128 V=8.0
MOVL C01129 V=8.0
MOVL C01130 V=8.0
MOVL C01131 V=8.0
MOVL C01132 V=8.0
MOVL C01133 V=8.0
MOVL C01134 V=8.0
MOVL C01135 V=8.0
MOVL C01136 V=8.0
MOVL C01137 V=8.0
MOVL C01138 V=8.0
MOVL C01139 V=8.0
MOVL C01140 V=8.0
MOVL C01141 V=8.0
MOVL C01142 V=8.0
MOVL C01143 V=8.0
MOVL C01144 V=8.0
MOVL C01145 V=8.0
MOVL C01146 V=8.0
MOVL C01147 V=8.0
MOVL C01148 V=8.0
MOVL C01149 V=8.0
MOVL C01150 V=8.0
MOVL C01151 V=8.0
MOVL C01152 V=8.0
MOVL C01153 V=8.0
MOVL C01154 V=8.0
MOVL C01155 V=8.0
MOVL C01156 V=8.0
MOVL C01157 V=8.0
MOVL C01158 V=8.0
MOVL C01159 V=8.0
MOVL C01160 V=8.0
MOVL C01161 V=8.0
MOVL C01162 V=8.0
MOVL C01163 V=8.0
MOVL C01164 V=8.0
MOVL C01165 V=8.0
MOVL C01166 V=8.0
MOVL C01167 V=8.0
MOVL C01168 V=8.0
MOVL C01169 V=8.0
MOVL C01170 V=8.0
MOVL C01171 V=8.0
MOVL C01172 V=8.0
MOVL C01173 V=8.0
MOVL C01174 V=8.0
MOVL C01175 V=8.0
MOVL C01176 V=8.0
MOVL C01177 V=8.0
MOVL C01178 V=8.0
MOVL C01179 V=8.0
MOVL C01180 V=8.0
MOVL C01181 V=8.0
MOVJ C01182 VJ=0.78
MOVL C01183 V=8.0
MOVL C01184 V=8.0
MOVL C01185 V=8.0
MOVL C01186 V=8.0
MOVL C01187 V=8.0
MOVL C01188 V=8.0
MOVL C01189 V=8.0
MOVL C01190 V=8.0
MOVL C01191 V=8.0
MOVL C01192 V=8.0
MOVL C01193 V=8.0
MOVL C01194 V=8.0
MOVL C01195 V=8.0
MOVL C01196 V=8.0
MOVL C01197 V=8.0
MOVL C01198 V=8.0
MOVL C01199 V=8.0
MOVL C01200 V=8.0
MOVL C01201 V=8.0
MOVL C01202 V=8.0
MOVL C01203 V=8.0
MOVL C01204 V=8.0
MOVL C01205 V=8.0
MOVL C01206 V=8.0
MOVL C01207 V=8.0
MOVL C01208 V=8.0
MOVL C01209 V=8.0
MOVL C01210 V=8.0
MOVL C01211 V=8.0
MOVL C01212 V=8.0
MOVL C01213 V=8.0
MOVL C01214 V=8.0
MOVL C01215 V=8.0
MOVL C01216 V=8.0
MOVL C01217 V=8.0
MOVL C01218 V=8.0
MOVL C01219 V=8.0
MOVL C01220 V=8.0
MOVL C01221 V=8.0
MOVL C01222 V=8.0
MOVL C01223 V=8.0
MOVJ C01224 VJ=0.78
MOVJ C01225 VJ=0.78
MOVL C01226 V=11.7
TIMER T=2.00
MOVL C01227 V=11.7
MOVJ C01228 VJ=0.78
MOVJ C01229 VJ=0.78
MOVL C01230 V=8.0
MOVL C01231 V=8.0
MOVL C01232 V=8.0
MOVL C01233 V=8.0
MOVL C01234 V=8.0
MOVL C01235 V=8.0
MOVL C01236 V=8.0
MOVL C01237 V=8.0
MOVL C01238 V=8.0
MOVL C01239 V=8.0
MOVL C01240 V=8.0
MOVL C01241 V=8.0
MOVL C01242 V=8.0
MOVL C01243 V=8.0
MOVL C01244 V=8.0
MOVL C01245 V=8.0
MOVL C01246 V=8.0
MOVL C01247 V=8.0
MOVL C01248 V=8.0
MOVL C01249 V=8.0
MOVL C01250 V=8.0
MOVL C01251 V=8.0
MOVJ C01252 VJ=0.78
MOVL C01253 V=8.0
MOVL C01254 V=8.0
MOVL C01255 V=8.0
MOVL C01256 V=8.0
MOVL C01257 V=8.0
MOVL C01258 V=8.0
MOVL C01259 V=8.0
MOVL C01260 V=8.0
MOVL C01261 V=8.0
MOVL C01262 V=8.0
MOVL C01263 V=8.0
MOVL C01264 V=8.0
MOVL C01265 V=8.0
MOVL C01266 V=8.0
MOVL C01267 V=8.0
MOVL C01268 V=8.0
MOVL C01269 V=8.0
MOVL C01270 V=8.0
MOVL C01271 V=8.0
MOVL C01272 V=8.0
MOVL C01273 V=8.0
MOVL C01274 V=8.0
MOVL C01275 V=8.0
MOVL C01276 V=8.0
MOVL C01277 V=8.0
MOVL C01278 V=8.0
MOVL C01279 V=8.0
MOVL C01280 V=8.0
MOVL C01281 V=8.0
MOVL C01282 V=8.0
MOVL C01283 V=8.0
MOVL C01284 V=8.0
MOVL C01285 V=8.0
MOVL C01286 V=8.0
MOVL C01287 V=8.0
MOVL C01288 V=8.0
MOVL C01289 V=8.0
MOVL C01290 V=8.0
MOVL C01291 V=8.0
MOVL C01292 V=8.0
MOVL C01293 V=8.0
MOVL C01294 V=8.0
MOVL C01295 V=8.0
MOVL C01296 V=8.0
MOVL C01297 V=8.0
MOVL C01298 V=8.0
MOVL C01299 V=8.0
MOVL C01300 V=8.0
MOVL C01301 V=8.0
MOVL C01302 V=8.0
MOVL C01303 V=8.0
MOVL C01304 V=8.0
MOVL C01305 V=8.0
MOVL C01306 V=8.0
MOVL C01307 V=8.0
MOVL C01308 V=8.0
MOVL C01309 V=8.0
MOVL C01310 V=8.0
MOVL C01311 V=8.0
MOVL C01312 V=8.0
MOVL C01313 V=8.0
MOVL C01314 V=8.0
MOVJ C01315 VJ=0.78
MOVL C01316 V=8.0
MOVL C01317 V=8.0
MOVL C01318 V=8.0
MOVL C01319 V=8.0
MOVL C01320 V=8.0
MOVL C01321 V=8.0
MOVL C01322 V=8.0
MOVL C01323 V=8.0
MOVL C01324 V=8.0
MOVL C01325 V=8.0
MOVL C01326 V=8.0
MOVL C01327 V=8.0
MOVL C01328 V=8.0
MOVL C01329 V=8.0
MOVL C01330 V=8.0
MOVL C01331 V=8.0
MOVL C01332 V=8.0
MOVL C01333 V=8.0
MOVL C01334 V=8.0
MOVL C01335 V=8.0
MOVL C01336 V=8.0
MOVL C01337 V=8.0
MOVL C01338 V=8.0
MOVL C01339 V=8.0
MOVL C01340 V=8.0
MOVL C01341 V=8.0
MOVL C01342 V=8.0
MOVL C01343 V=8.0
MOVL C01344 V=8.0
MOVL C01345 V=8.0
MOVL C01346 V=8.0
MOVL C01347 V=8.0
MOVL C01348 V=8.0
MOVL C01349 V=8.0
MOVL C01350 V=8.0
MOVL C01351 V=8.0
MOVL C01352 V=8.0
MOVL C01353 V=8.0
MOVL C01354 V=8.0
MOVL C01355 V=8.0
MOVL C01356 V=8.0
MOVL C01357 V=8.0
MOVL C01358 V=8.0
MOVL C01359 V=8.0
MOVL C01360 V=8.0
MOVL C01361 V=8.0
MOVL C01362 V=8.0
MOVL C01363 V=8.0
MOVL C01364 V=8.0
MOVL C01365 V=8.0
MOVL C01366 V=8.0
MOVL C01367 V=8.0
MOVL C01368 V=8.0
MOVL C01369 V=8.0
MOVL C01370 V=8.0
MOVL C01371 V=8.0
MOVL C01372 V=8.0
MOVL C01373 V=8.0
MOVL C01374 V=8.0
MOVL C01375 V=8.0
MOVL C01376 V=8.0
MOVL C01377 V=8.0
MOVJ C01378 VJ=0.78
MOVL C01379 V=8.0
MOVL C01380 V=8.0
MOVL C01381 V=8.0
MOVL C01382 V=8.0
MOVL C01383 V=8.0
MOVL C01384 V=8.0
MOVL C01385 V=8.0
MOVL C01386 V=8.0
MOVL C01387 V=8.0
MOVL C01388 V=8.0
MOVL C01389 V=8.0
MOVL C01390 V=8.0
MOVL C01391 V=8.0
MOVL C01392 V=8.0
MOVL C01393 V=8.0
MOVL C01394 V=8.0
MOVL C01395 V=8.0
MOVL C01396 V=8.0
MOVL C01397 V=8.0
MOVL C01398 V=8.0
MOVL C01399 V=8.0
MOVJ C01400 VJ=0.78
MOVJ C01401 VJ=0.78
MOVL C01402 V=11.7
TIMER T=2.00
MOVL C01403 V=11.7
MOVJ C01404 VJ=0.78
MOVJ C01405 VJ=0.78
MOVL C01406 V=8.0
MOVL C01407 V=8.0
MOVL C01408 V=8.0
MOVL C01409 V=8.0
MOVL C01410 V=8.0
MOVL C01411 V=8.0
MOVL C01412 V=8.0
MOVL C01413 V=8.0
MOVL C01414 V=8.0
MOVL C01415 V=8.0
MOVL C01416 V=8.0
MOVL C01417 V=8.0
MOVL C01418 V=8.0
MOVL C01419 V=8.0
MOVL C01420 V=8.0
MOVL C01421 V=8.0
MOVL C01422 V=8.0
MOVL C01423 V=8.0
MOVL C01424 V=8.0
MOVL C01425 V=8.0
MOVL C01426 V=8.0
MOVL C01427 V=8.0
MOVL C01428 V=8.0
MOVL C01429 V=8.0
MOVL C01430 V=8.0
MOVL C01431 V=8.0
MOVL C01432 V=8.0
MOVL C01433 V=8.0
MOVL C01434 V=8.0
MOVL C01435 V=8.0
MOVL C01436 V=8.0
MOVL C01437 V=8.0
MOVL C01438 V=8.0
MOVL C01439 V=8.0
MOVL C01440 V=8.0
MOVL C01441 V=8.0
MOVL C01442 V=8.0
MOVL C01443 V=8.0
MOVL C01444 V=8.0
MOVL C01445 V=8.0
MOVL C01446 V=8.0
MOVL C01447 V=8.0
MOVJ C01448 VJ=0.78
MOVL C01449 V=8.0
MOVL C01450 V=8.0
MOVL C01451 V=8.0
MOVL C01452 V=8.0
MOVL C01453 V=8.0
MOVL C01454 V=8.0
MOVL C01455 V=8.0
MOVL C01456 V=8.0
MOVL C01457 V=8.0
MOVL C01458 V=8.0
MOVL C01459 V=8.0
MOVL C01460 V=8.0
MOVL C01461 V=8.0
MOVL C01462 V=8.0
MOVL C01463 V=8.0
MOVL C01464 V=8.0
MOVL C01465 V=8.0
MOVL C01466 V=8.0
MOVL C01467 V=8.0
MOVL C01468 V=8.0
MOVL C01469 V=8.0
MOVL C01470 V=8.0
MOVL C01471 V=8.0
MOVL C01472 V=8.0
MOVL C01473 V=8.0
MOVL C01474 V=8.0
MOVL C01475 V=8.0
MOVL C01476 V=8.0
MOVL C01477 V=8.0
MOVL C01478 V=8.0
MOVL C01479 V=8.0
MOVL C01480 V=8.0
MOVL C01481 V=8.0
MOVL C01482 V=8.0
MOVL C01483 V=8.0
MOVL C01484 V=8.0
MOVL C01485 V=8.0
MOVL C01486 V=8.0
MOVL C01487 V=8.0
MOVL C01488 V=8.0
MOVL C01489 V=8.0
MOVL C01490 V=8.0
MOVL C01491 V=8.0
MOVL C01492 V=8.0
MOVL C01493 V=8.0
MOVL C01494 V=8.0
MOVL C01495 V=8.0
MOVL C01496 V=8.0
MOVL C01497 V=8.0
MOVL C01498 V=8.0
MOVL C01499 V=8.0
MOVL C01500 V=8.0
MOVL C01501 V=8.0
MOVL C01502 V=8.0
MOVL C01503 V=8.0
MOVL C01504 V=8.0
MOVL C01505 V=8.0
MOVL C01506 V=8.0
MOVL C01507 V=8.0
MOVL C01508 V=8.0
MOVL C01509 V=8.0
MOVL C01510 V=8.0
MOVJ C01511 VJ=0.78
MOVL C01512 V=8.0
MOVL C01513 V=8.0
MOVL C01514 V=8.0
MOVL C01515 V=8.0
MOVL C01516 V=8.0
MOVL C01517 V=8.0
MOVL C01518 V=8.0
MOVL C01519 V=8.0
MOVL C01520 V=8.0
MOVL C01521 V=8.0
MOVL C01522 V=8.0
MOVL C01523 V=8.0
MOVL C01524 V=8.0
MOVL C01525 V=8.0
MOVL C01526 V=8.0
MOVL C01527 V=8.0
MOVL C01528 V=8.0
MOVL C01529 V=8.0
MOVL C01530 V=8.0
MOVL C01531 V=8.0
MOVL C01532 V=8.0
MOVL C01533 V=8.0
MOVL C01534 V=8.0
MOVL C01535 V=8.0
MOVL C01536 V=8.0
MOVL C01537 V=8.0
MOVL C01538 V=8.0
MOVL C01539 V=8.0
MOVL C01540 V=8.0
MOVL C01541 V=8.0
MOVL C01542 V=8.0
MOVL C01543 V=8.0
MOVL C01544 V=8.0
MOVL C01545 V=8.0
MOVL C01546 V=8.0
MOVL C01547 V=8.0
MOVL C01548 V=8.0
MOVL C01549 V=8.0
MOVL C01550 V=8.0
MOVL C01551 V=8.0
MOVL C01552 V=8.0
MOVL C01553 V=8.0
MOVL C01554 V=8.0
MOVL C01555 V=8.0
MOVL C01556 V=8.0
MOVL C01557 V=8.0
MOVL C01558 V=8.0
MOVL C01559 V=8.0
MOVL C01560 V=8.0
MOVL C01561 V=8.0
MOVL C01562 V=8.0
MOVL C01563 V=8.0
MOVL C01564 V=8.0
MOVL C01565 V=8.0
MOVL C01566 V=8.0
MOVL C01567 V=8.0
MOVL C01568 V=8.0
MOVL C01569 V=8.0
MOVL C01570 V=8.0
MOVL C01571 V=8.0
MOVL C01572 V=8.0
MOVJ C01573 VJ=0.78
MOVJ C01574 VJ=0.78
MOVL C01575 V=11.7
TIMER T=2.00
MOVL C01576 V=11.7
MOVJ C01577 VJ=0.78
MOVJ C01578 VJ=0.78
MOVL C01579 V=8.0
MOVL C01580 V=8.0
MOVJ C01581 VJ=0.78
MOVL C01582 V=8.0
MOVL C01583 V=8.0
MOVL C01584 V=8.0
MOVL C01585 V=8.0
MOVL C01586 V=8.0
MOVL C01587 V=8.0
MOVL C01588 V=8.0
MOVL C01589 V=8.0
MOVL C01590 V=8.0
MOVL C01591 V=8.0
MOVL C01592 V=8.0
MOVL C01593 V=8.0
MOVL C01594 V=8.0
MOVL C01595 V=8.0
MOVL C01596 V=8.0
MOVL C01597 V=8.0
MOVL C01598 V=8.0
MOVL C01599 V=8.0
MOVL C01600 V=8.0
MOVL C01601 V=8.0
MOVL C01602 V=8.0
MOVL C01603 V=8.0
MOVL C01604 V=8.0
MOVL C01605 V=8.0
MOVL C01606 V=8.0
MOVL C01607 V=8.0
MOVL C01608 V=8.0
MOVL C01609 V=8.0
MOVL C01610 V=8.0
MOVL C01611 V=8.0
MOVL C01612 V=8.0
MOVL C01613 V=8.0
MOVL C01614 V=8.0
MOVL C01615 V=8.0
MOVL C01616 V=8.0
MOVL C01617 V=8.0
MOVL C01618 V=8.0
MOVL C01619 V=8.0
MOVL C01620 V=8.0
MOVL C01621 V=8.0
MOVL C01622 V=8.0
MOVL C01623 V=8.0
MOVL C01624 V=8.0
MOVL C01625 V=8.0
MOVL C01626 V=8.0
MOVL C01627 V=8.0
MOVL C01628 V=8.0
MOVL C01629 V=8.0
MOVL C01630 V=8.0
MOVL C01631 V=8.0
MOVL C01632 V=8.0
MOVL C01633 V=8.0
MOVL C01634 V=8.0
MOVL C01635 V=8.0
MOVL C01636 V=8.0
MOVL C01637 V=8.0
MOVL C01638 V=8.0
MOVL C01639 V=8.0
MOVL C01640 V=8.0
MOVL C01641 V=8.0
MOVL C01642 V=8.0
MOVL C01643 V=8.0
MOVJ C01644 VJ=0.78
MOVL C01645 V=8.0
MOVL C01646 V=8.0
MOVL C01647 V=8.0
MOVL C01648 V=8.0
MOVL C01649 V=8.0
MOVL C01650 V=8.0
MOVL C01651 V=8.0
MOVL C01652 V=8.0
MOVL C01653 V=8.0
MOVL C01654 V=8.0
MOVL C01655 V=8.0
MOVL C01656 V=8.0
MOVL C01657 V=8.0
MOVL C01658 V=8.0
MOVL C01659 V=8.0
MOVL C01660 V=8.0
MOVL C01661 V=8.0
MOVL C01662 V=8.0
MOVL C01663 V=8.0
MOVL C01664 V=8.0
MOVL C01665 V=8.0
MOVL C01666 V=8.0
MOVL C01667 V=8.0
MOVL C01668 V=8.0
MOVL C01669 V=8.0
MOVL C01670 V=8.0
MOVL C01671 V=8.0
MOVL C01672 V=8.0
MOVL C01673 V=8.0
MOVL C01674 V=8.0
MOVL C01675 V=8.0
MOVL C01676 V=8.0
MOVL C01677 V=8.0
MOVL C01678 V=8.0
MOVL C01679 V=8.0
MOVL C01680 V=8.0
MOVL C01681 V=8.0
MOVL C01682 V=8.0
MOVL C01683 V=8.0
MOVL C01684 V=8.0
MOVL C01685 V=8.0
MOVL C01686 V=8.0
MOVL C01687 V=8.0
MOVL C01688 V=8.0
MOVL C01689 V=8.0
MOVL C01690 V=8.0
MOVL C01691 V=8.0
MOVL C01692 V=8.0
MOVL C01693 V=8.0
MOVL C01694 V=8.0
MOVL C01695 V=8.0
MOVL C01696 V=8.0
MOVL C01697 V=8.0
MOVL C01698 V=8.0
MOVL C01699 V=8.0
MOVL C01700 V=8.0
MOVL C01701 V=8.0
MOVL C01702 V=8.0
MOVL C01703 V=8.0
MOVL C01704 V=8.0
MOVL C01705 V=8.0
MOVL C01706 V=8.0
MOVJ C01707 VJ=0.78
MOVL C01708 V=8.0
MOVL C01709 V=8.0
MOVL C01710 V=8.0
MOVL C01711 V=8.0
MOVL C01712 V=8.0
MOVL C01713 V=8.0
MOVL C01714 V=8.0
MOVL C01715 V=8.0
MOVL C01716 V=8.0
MOVL C01717 V=8.0
MOVL C01718 V=8.0
MOVL C01719 V=8.0
MOVL C01720 V=8.0
MOVL C01721 V=8.0
MOVL C01722 V=8.0
MOVL C01723 V=8.0
MOVL C01724 V=8.0
MOVL C01725 V=8.0
MOVL C01726 V=8.0
MOVL C01727 V=8.0
MOVL C01728 V=8.0
MOVL C01729 V=8.0
MOVL C01730 V=8.0
MOVL C01731 V=8.0
MOVL C01732 V=8.0
MOVL C01733 V=8.0
MOVL C01734 V=8.0
MOVL C01735 V=8.0
MOVL C01736 V=8.0
MOVL C01737 V=8.0
MOVL C01738 V=8.0
MOVL C01739 V=8.0
MOVL C01740 V=8.0
MOVL C01741 V=8.0
MOVL C01742 V=8.0
MOVL C01743 V=8.0
MOVL C01744 V=8.0
MOVL C01745 V=8.0
MOVL C01746 V=8.0
MOVL C01747 V=8.0
MOVL C01748 V=8.0
MOVJ C01749 VJ=0.78
MOVJ C01750 VJ=0.78
MOVL C01751 V=11.7
TIMER T=2.00
MOVL C01752 V=11.7
MOVJ C01753 VJ=0.78
MOVJ C01754 VJ=0.78
MOVL C01755 V=8.0
MOVL C01756 V=8.0
MOVL C01757 V=8.0
MOVL C01758 V=8.0
MOVL C01759 V=8.0
MOVL C01760 V=8.0
MOVL C01761 V=8.0
MOVL C01762 V=8.0
MOVL C01763 V=8.0
MOVL C01764 V=8.0
MOVL C01765 V=8.0
MOVL C01766 V=8.0
MOVL C01767 V=8.0
MOVL C01768 V=8.0
MOVL C01769 V=8.0
MOVL C01770 V=8.0
MOVL C01771 V=8.0
MOVL C01772 V=8.0
MOVL C01773 V=8.0
MOVL C01774 V=8.0
MOVL C01775 V=8.0
MOVL C01776 V=8.0
MOVJ C01777 VJ=0.78
MOVL C01778 V=8.0
MOVL C01779 V=8.0
MOVL C01780 V=8.0
MOVL C01781 V=8.0
MOVL C01782 V=8.0
MOVL C01783 V=8.0
MOVL C01784 V=8.0
MOVL C01785 V=8.0
MOVL C01786 V=8.0
MOVL C01787 V=8.0
MOVL C01788 V=8.0
MOVL C01789 V=8.0
MOVL C01790 V=8.0
MOVL C01791 V=8.0
MOVL C01792 V=8.0
MOVL C01793 V=8.0
MOVL C01794 V=8.0
MOVL C01795 V=8.0
MOVL C01796 V=8.0
MOVL C01797 V=8.0
MOVL C01798 V=8.0
MOVL C01799 V=8.0
MOVL C01800 V=8.0
MOVL C01801 V=8.0
MOVL C01802 V=8.0
MOVL C01803 V=8.0
MOVL C01804 V=8.0
MOVL C01805 V=8.0
MOVL C01806 V=8.0
MOVL C01807 V=8.0
MOVL C01808 V=8.0
MOVL C01809 V=8.0
MOVL C01810 V=8.0
MOVL C01811 V=8.0
MOVL C01812 V=8.0
MOVL C01813 V=8.0
MOVL C01814 V=8.0
MOVL C01815 V=8.0
MOVL C01816 V=8.0
MOVL C01817 V=8.0
MOVL C01818 V=8.0
MOVL C01819 V=8.0
MOVL C01820 V=8.0
MOVL C01821 V=8.0
MOVL C01822 V=8.0
MOVL C01823 V=8.0
MOVL C01824 V=8.0
MOVL C01825 V=8.0
MOVL C01826 V=8.0
MOVL C01827 V=8.0
MOVL C01828 V=8.0
MOVL C01829 V=8.0
MOVL C01830 V=8.0
MOVL C01831 V=8.0
MOVL C01832 V=8.0
MOVL C01833 V=8.0
MOVL C01834 V=8.0
MOVL C01835 V=8.0
MOVL C01836 V=8.0
MOVL C01837 V=8.0
MOVL C01838 V=8.0
MOVL C01839 V=8.0
MOVJ C01840 VJ=0.78
MOVL C01841 V=8.0
MOVL C01842 V=8.0
MOVL C01843 V=8.0
MOVL C01844 V=8.0
MOVL C01845 V=8.0
MOVL C01846 V=8.0
MOVL C01847 V=8.0
MOVL C01848 V=8.0
MOVL C01849 V=8.0
MOVL C01850 V=8.0
MOVL C01851 V=8.0
MOVL C01852 V=8.0
MOVL C01853 V=8.0
MOVL C01854 V=8.0
MOVL C01855 V=8.0
MOVL C01856 V=8.0
MOVL C01857 V=8.0
MOVL C01858 V=8.0
MOVL C01859 V=8.0
MOVL C01860 V=8.0
MOVL C01861 V=8.0
MOVL C01862 V=8.0
MOVL C01863 V=8.0
MOVL C01864 V=8.0
MOVL C01865 V=8.0
MOVL C01866 V=8.0
MOVL C01867 V=8.0
MOVL C01868 V=8.0
MOVL C01869 V=8.0
MOVL C01870 V=8.0
MOVL C01871 V=8.0
MOVL C01872 V=8.0
MOVL C01873 V=8.0
MOVL C01874 V=8.0
MOVL C01875 V=8.0
MOVL C01876 V=8.0
MOVL C01877 V=8.0
MOVL C01878 V=8.0
MOVL C01879 V=8.0
MOVL C01880 V=8.0
MOVL C01881 V=8.0
MOVL C01882 V=8.0
MOVL C01883 V=8.0
MOVL C01884 V=8.0
MOVL C01885 V=8.0
MOVL C01886 V=8.0
MOVL C01887 V=8.0
MOVL C01888 V=8.0
MOVL C01889 V=8.0
MOVL C01890 V=8.0
MOVL C01891 V=8.0
MOVL C01892 V=8.0
MOVL C01893 V=8.0
MOVL C01894 V=8.0
MOVL C01895 V=8.0
MOVL C01896 V=8.0
MOVL C01897 V=8.0
MOVL C01898 V=8.0
MOVL C01899 V=8.0
MOVL C01900 V=8.0
MOVL C01901 V=8.0
MOVL C01902 V=8.0
MOVJ C01903 VJ=0.78
MOVL C01904 V=8.0
MOVL C01905 V=8.0
MOVL C01906 V=8.0
MOVL C01907 V=8.0
MOVL C01908 V=8.0
MOVL C01909 V=8.0
MOVL C01910 V=8.0
MOVL C01911 V=8.0
MOVL C01912 V=8.0
MOVL C01913 V=8.0
MOVL C01914 V=8.0
MOVL C01915 V=8.0
MOVL C01916 V=8.0
MOVL C01917 V=8.0
MOVL C01918 V=8.0
MOVL C01919 V=8.0
MOVL C01920 V=8.0
MOVL C01921 V=8.0
MOVL C01922 V=8.0
MOVL C01923 V=8.0
MOVL C01924 V=8.0
MOVJ C01925 VJ=0.78
MOVJ C01926 VJ=0.78
MOVL C01927 V=11.7
TIMER T=2.00
MOVL C01928 V=11.7
MOVJ C01929 VJ=0.78
MOVJ C01930 VJ=0.78
MOVL C01931 V=8.0
MOVL C01932 V=8.0
MOVL C01933 V=8.0
MOVL C01934 V=8.0
MOVL C01935 V=8.0
MOVL C01936 V=8.0
MOVL C01937 V=8.0
MOVL C01938 V=8.0
MOVL C01939 V=8.0
MOVL C01940 V=8.0
MOVL C01941 V=8.0
MOVL C01942 V=8.0
MOVL C01943 V=8.0
MOVL C01944 V=8.0
MOVL C01945 V=8.0
MOVL C01946 V=8.0
MOVL C01947 V=8.0
MOVL C01948 V=8.0
MOVL C01949 V=8.0
MOVL C01950 V=8.0
MOVL C01951 V=8.0
MOVL C01952 V=8.0
MOVL C01953 V=8.0
MOVL C01954 V=8.0
MOVL C01955 V=8.0
MOVL C01956 V=8.0
MOVL C01957 V=8.0
MOVL C01958 V=8.0
MOVL C01959 V=8.0
MOVL C01960 V=8.0
MOVL C01961 V=8.0
MOVL C01962 V=8.0
MOVL C01963 V=8.0
MOVL C01964 V=8.0
MOVL C01965 V=8.0
MOVL C01966 V=8.0
MOVL C01967 V=8.0
MOVL C01968 V=8.0
MOVL C01969 V=8.0
MOVL C01970 V=8.0
MOVL C01971 V=8.0
MOVL C01972 V=8.0
MOVJ C01973 VJ=0.78
MOVL C01974 V=8.0
MOVL C01975 V=8.0
MOVL C01976 V=8.0
MOVL C01977 V=8.0
MOVL C01978 V=8.0
MOVL C01979 V=8.0
MOVL C01980 V=8.0
MOVL C01981 V=8.0
MOVL C01982 V=8.0
MOVL C01983 V=8.0
MOVL C01984 V=8.0
MOVL C01985 V=8.0
MOVL C01986 V=8.0
MOVL C01987 V=8.0
MOVL C01988 V=8.0
MOVL C01989 V=8.0
MOVL C01990 V=8.0
MOVL C01991 V=8.0
MOVL C01992 V=8.0
MOVL C01993 V=8.0
MOVL C01994 V=8.0
MOVL C01995 V=8.0
MOVL C01996 V=8.0
MOVL C01997 V=8.0
MOVL C01998 V=8.0
MOVL C01999 V=8.0
MOVL C02000 V=8.0
MOVL C02001 V=8.0
MOVL C02002 V=8.0
MOVL C02003 V=8.0
MOVL C02004 V=8.0
MOVL C02005 V=8.0
MOVL C02006 V=8.0
MOVL C02007 V=8.0
MOVL C02008 V=8.0
MOVL C02009 V=8.0
MOVL C02010 V=8.0
MOVL C02011 V=8.0
MOVL C02012 V=8.0
MOVL C02013 V=8.0
MOVL C02014 V=8.0
MOVL C02015 V=8.0
MOVL C02016 V=8.0
MOVL C02017 V=8.0
MOVL C02018 V=8.0
MOVL C02019 V=8.0
MOVL C02020 V=8.0
MOVL C02021 V=8.0
MOVL C02022 V=8.0
MOVL C02023 V=8.0
MOVL C02024 V=8.0
MOVL C02025 V=8.0
MOVL C02026 V=8.0
MOVL C02027 V=8.0
MOVL C02028 V=8.0
MOVL C02029 V=8.0
MOVL C02030 V=8.0
MOVL C02031 V=8.0
MOVL C02032 V=8.0
MOVL C02033 V=8.0
MOVL C02034 V=8.0
MOVL C02035 V=8.0
MOVJ C02036 VJ=0.78
MOVL C02037 V=8.0
MOVL C02038 V=8.0
MOVL C02039 V=8.0
MOVL C02040 V=8.0
MOVL C02041 V=8.0
MOVL C02042 V=8.0
MOVL C02043 V=8.0
MOVL C02044 V=8.0
MOVL C02045 V=8.0
MOVL C02046 V=8.0
MOVL C02047 V=8.0
MOVL C02048 V=8.0
MOVL C02049 V=8.0
MOVL C02050 V=8.0
MOVL C02051 V=8.0
MOVL C02052 V=8.0
MOVL C02053 V=8.0
MOVL C02054 V=8.0
MOVL C02055 V=8.0
MOVL C02056 V=8.0
MOVL C02057 V=8.0
MOVL C02058 V=8.0
MOVL C02059 V=8.0
MOVL C02060 V=8.0
MOVL C02061 V=8.0
MOVL C02062 V=8.0
MOVL C02063 V=8.0
MOVL C02064 V=8.0
MOVL C02065 V=8.0
MOVL C02066 V=8.0
MOVL C02067 V=8.0
MOVL C02068 V=8.0
MOVL C02069 V=8.0
MOVL C02070 V=8.0
MOVL C02071 V=8.0
MOVL C02072 V=8.0
MOVL C02073 V=8.0
MOVL C02074 V=8.0
MOVL C02075 V=8.0
MOVL C02076 V=8.0
MOVL C02077 V=8.0
MOVL C02078 V=8.0
MOVL C02079 V=8.0
MOVL C02080 V=8.0
MOVL C02081 V=8.0
MOVL C02082 V=8.0
MOVL C02083 V=8.0
MOVL C02084 V=8.0
MOVL C02085 V=8.0
MOVL C02086 V=8.0
MOVL C02087 V=8.0
MOVL C02088 V=8.0
MOVL C02089 V=8.0
MOVL C02090 V=8.0
MOVL C02091 V=8.0
MOVL C02092 V=8.0
MOVL C02093 V=8.0
MOVL C02094 V=8.0
MOVL C02095 V=8.0
MOVL C02096 V=8.0
MOVL C02097 V=8.0
MOVJ C02098 VJ=0.78
MOVJ C02099 VJ=0.78
MOVL C02100 V=11.7
TIMER T=2.00
MOVL C02101 V=11.7
MOVJ C02102 VJ=0.78
MOVJ C02103 VJ=0.78
MOVL C02104 V=8.0
MOVL C02105 V=8.0
MOVJ C02106 VJ=0.78
MOVL C02107 V=8.0
MOVL C02108 V=8.0
MOVL C02109 V=8.0
MOVL C02110 V=8.0
MOVL C02111 V=8.0
MOVL C02112 V=8.0
MOVL C02113 V=8.0
MOVL C02114 V=8.0
MOVL C02115 V=8.0
MOVL C02116 V=8.0
MOVL C02117 V=8.0
MOVL C02118 V=8.0
MOVL C02119 V=8.0
MOVL C02120 V=8.0
MOVL C02121 V=8.0
MOVL C02122 V=8.0
MOVL C02123 V=8.0
MOVL C02124 V=8.0
MOVL C02125 V=8.0
MOVL C02126 V=8.0
MOVL C02127 V=8.0
MOVL C02128 V=8.0
MOVL C02129 V=8.0
MOVL C02130 V=8.0
MOVL C02131 V=8.0
MOVL C02132 V=8.0
MOVL C02133 V=8.0
MOVL C02134 V=8.0
MOVL C02135 V=8.0
MOVL C02136 V=8.0
MOVL C02137 V=8.0
MOVL C02138 V=8.0
MOVL C02139 V=8.0
MOVL C02140 V=8.0
MOVL C02141 V=8.0
MOVL C02142 V=8.0
MOVL C02143 V=8.0
MOVL C02144 V=8.0
MOVL C02145 V=8.0
MOVL C02146 V=8.0
MOVL C02147 V=8.0
MOVL C02148 V=8.0
MOVL C02149 V=8.0
MOVL C02150 V=8.0
MOVL C02151 V=8.0
MOVL C02152 V=8.0
MOVL C02153 V=8.0
MOVL C02154 V=8.0
MOVL C02155 V=8.0
MOVL C02156 V=8.0
MOVL C02157 V=8.0
MOVL C02158 V=8.0
MOVL C02159 V=8.0
MOVL C02160 V=8.0
MOVL C02161 V=8.0
MOVL C02162 V=8.0
MOVL C02163 V=8.0
MOVL C02164 V=8.0
MOVL C02165 V=8.0
MOVL C02166 V=8.0
MOVL C02167 V=8.0
MOVL C02168 V=8.0
MOVJ C02169 VJ=0.78
MOVL C02170 V=8.0
MOVL C02171 V=8.0
MOVL C02172 V=8.0
MOVL C02173 V=8.0
MOVL C02174 V=8.0
MOVL C02175 V=8.0
MOVL C02176 V=8.0
MOVL C02177 V=8.0
MOVL C02178 V=8.0
MOVL C02179 V=8.0
MOVL C02180 V=8.0
MOVL C02181 V=8.0
MOVL C02182 V=8.0
MOVL C02183 V=8.0
MOVL C02184 V=8.0
MOVL C02185 V=8.0
MOVL C02186 V=8.0
MOVL C02187 V=8.0
MOVL C02188 V=8.0
MOVL C02189 V=8.0
MOVL C02190 V=8.0
MOVL C02191 V=8.0
MOVL C02192 V=8.0
MOVL C02193 V=8.0
MOVL C02194 V=8.0
MOVL C02195 V=8.0
MOVL C02196 V=8.0
MOVL C02197 V=8.0
MOVL C02198 V=8.0
MOVL C02199 V=8.0
MOVL C02200 V=8.0
MOVL C02201 V=8.0
MOVL C02202 V=8.0
MOVL C02203 V=8.0
MOVL C02204 V=8.0
MOVL C02205 V=8.0
MOVL C02206 V=8.0
MOVL C02207 V=8.0
MOVL C02208 V=8.0
MOVL C02209 V=8.0
MOVL C02210 V=8.0
MOVL C02211 V=8.0
MOVL C02212 V=8.0
MOVL C02213 V=8.0
MOVL C02214 V=8.0
MOVL C02215 V=8.0
MOVL C02216 V=8.0
MOVL C02217 V=8.0
MOVL C02218 V=8.0
MOVL C02219 V=8.0
MOVL C02220 V=8.0
MOVL C02221 V=8.0
MOVL C02222 V=8.0
MOVL C02223 V=8.0
MOVL C02224 V=8.0
MOVL C02225 V=8.0
MOVL C02226 V=8.0
MOVL C02227 V=8.0
MOVL C02228 V=8.0
MOVL C02229 V=8.0
MOVL C02230 V=8.0
MOVL C02231 V=8.0
MOVJ C02232 VJ=0.78
MOVL C02233 V=8.0
MOVL C02234 V=8.0
MOVL C02235 V=8.0
MOVL C02236 V=8.0
MOVL C02237 V=8.0
MOVL C02238 V=8.0
MOVL C02239 V=8.0
MOVL C02240 V=8.0
MOVL C02241 V=8.0
MOVL C02242 V=8.0
MOVL C02243 V=8.0
MOVL C02244 V=8.0
MOVL C02245 V=8.0
MOVL C02246 V=8.0
MOVL C02247 V=8.0
MOVL C02248 V=8.0
MOVL C02249 V=8.0
MOVL C02250 V=8.0
MOVL C02251 V=8.0
MOVL C02252 V=8.0
MOVL C02253 V=8.0
MOVL C02254 V=8.0
MOVL C02255 V=8.0
MOVL C02256 V=8.0
MOVL C02257 V=8.0
MOVL C02258 V=8.0
MOVL C02259 V=8.0
MOVL C02260 V=8.0
MOVL C02261 V=8.0
MOVL C02262 V=8.0
MOVL C02263 V=8.0
MOVL C02264 V=8.0
MOVL C02265 V=8.0
MOVL C02266 V=8.0
MOVL C02267 V=8.0
MOVL C02268 V=8.0
MOVL C02269 V=8.0
MOVL C02270 V=8.0
MOVL C02271 V=8.0
MOVL C02272 V=8.0
MOVL C02273 V=8.0
MOVJ C02274 VJ=0.78
MOVJ C02275 VJ=0.78
MOVL C02276 V=11.7
TIMER T=2.00
MOVL C02277 V=11.7
MOVJ C02278 VJ=0.78
MOVJ C02279 VJ=0.78
MOVL C02280 V=8.0
MOVL C02281 V=8.0
MOVL C02282 V=8.0
MOVL C02283 V=8.0
MOVL C02284 V=8.0
MOVL C02285 V=8.0
MOVL C02286 V=8.0
MOVL C02287 V=8.0
MOVL C02288 V=8.0
MOVL C02289 V=8.0
MOVL C02290 V=8.0
MOVL C02291 V=8.0
MOVL C02292 V=8.0
MOVL C02293 V=8.0
MOVL C02294 V=8.0
MOVL C02295 V=8.0
MOVL C02296 V=8.0
MOVL C02297 V=8.0
MOVL C02298 V=8.0
MOVL C02299 V=8.0
MOVL C02300 V=8.0
MOVL C02301 V=8.0
MOVJ C02302 VJ=0.78
MOVL C02303 V=8.0
MOVL C02304 V=8.0
MOVL C02305 V=8.0
MOVL C02306 V=8.0
MOVL C02307 V=8.0
MOVL C02308 V=8.0
MOVL C02309 V=8.0
MOVL C02310 V=8.0
MOVL C02311 V=8.0
MOVL C02312 V=8.0
MOVL C02313 V=8.0
MOVL C02314 V=8.0
MOVL C02315 V=8.0
MOVL C02316 V=8.0
MOVL C02317 V=8.0
MOVL C02318 V=8.0
MOVL C02319 V=8.0
MOVL C02320 V=8.0
MOVL C02321 V=8.0
MOVL C02322 V=8.0
MOVL C02323 V=8.0
MOVL C02324 V=8.0
MOVL C02325 V=8.0
MOVL C02326 V=8.0
MOVL C02327 V=8.0
MOVL C02328 V=8.0
MOVL C02329 V=8.0
MOVL C02330 V=8.0
MOVL C02331 V=8.0
MOVL C02332 V=8.0
MOVL C02333 V=8.0
MOVL C02334 V=8.0
MOVL C02335 V=8.0
MOVL C02336 V=8.0
MOVL C02337 V=8.0
MOVL C02338 V=8.0
MOVL C02339 V=8.0
MOVL C02340 V=8.0
MOVL C02341 V=8.0
MOVL C02342 V=8.0
MOVL C02343 V=8.0
MOVL C02344 V=8.0
MOVL C02345 V=8.0
MOVL C02346 V=8.0
MOVL C02347 V=8.0
MOVL C02348 V=8.0
MOVL C02349 V=8.0
MOVL C02350 V=8.0
MOVL C02351 V=8.0
MOVL C02352 V=8.0
MOVL C02353 V=8.0
MOVL C02354 V=8.0
MOVL C02355 V=8.0
MOVL C02356 V=8.0
MOVL C02357 V=8.0
MOVL C02358 V=8.0
MOVL C02359 V=8.0
MOVL C02360 V=8.0
MOVL C02361 V=8.0
MOVL C02362 V=8.0
MOVL C02363 V=8.0
MOVL C02364 V=8.0
MOVJ C02365 VJ=0.78
MOVL C02366 V=8.0
MOVL C02367 V=8.0
MOVL C02368 V=8.0
MOVL C02369 V=8.0
MOVL C02370 V=8.0
MOVL C02371 V=8.0
MOVL C02372 V=8.0
MOVL C02373 V=8.0
MOVL C02374 V=8.0
MOVL C02375 V=8.0
MOVL C02376 V=8.0
MOVL C02377 V=8.0
MOVL C02378 V=8.0
MOVL C02379 V=8.0
MOVL C02380 V=8.0
MOVL C02381 V=8.0
MOVL C02382 V=8.0
MOVL C02383 V=8.0
MOVL C02384 V=8.0
MOVL C02385 V=8.0
MOVL C02386 V=8.0
MOVL C02387 V=8.0
MOVL C02388 V=8.0
MOVL C02389 V=8.0
MOVL C02390 V=8.0
MOVL C02391 V=8.0
MOVL C02392 V=8.0
MOVL C02393 V=8.0
MOVL C02394 V=8.0
MOVL C02395 V=8.0
MOVL C02396 V=8.0
MOVL C02397 V=8.0
MOVL C02398 V=8.0
MOVL C02399 V=8.0
MOVL C02400 V=8.0
MOVL C02401 V=8.0
MOVL C02402 V=8.0
MOVL C02403 V=8.0
MOVL C02404 V=8.0
MOVL C02405 V=8.0
MOVL C02406 V=8.0
MOVL C02407 V=8.0
MOVL C02408 V=8.0
MOVL C02409 V=8.0
MOVL C02410 V=8.0
MOVL C02411 V=8.0
MOVL C02412 V=8.0
MOVL C02413 V=8.0
MOVL C02414 V=8.0
MOVL C02415 V=8.0
MOVL C02416 V=8.0
MOVL C02417 V=8.0
MOVL C02418 V=8.0
MOVL C02419 V=8.0
MOVL C02420 V=8.0
MOVL C02421 V=8.0
MOVL C02422 V=8.0
MOVL C02423 V=8.0
MOVL C02424 V=8.0
MOVL C02425 V=8.0
MOVL C02426 V=8.0
MOVL C02427 V=8.0
MOVJ C02428 VJ=0.78
MOVL C02429 V=8.0
MOVL C02430 V=8.0
MOVL C02431 V=8.0
MOVL C02432 V=8.0
MOVL C02433 V=8.0
MOVL C02434 V=8.0
MOVL C02435 V=8.0
MOVL C02436 V=8.0
MOVL C02437 V=8.0
MOVL C02438 V=8.0
MOVL C02439 V=8.0
MOVL C02440 V=8.0
MOVL C02441 V=8.0
MOVL C02442 V=8.0
MOVL C02443 V=8.0
MOVL C02444 V=8.0
MOVL C02445 V=8.0
MOVL C02446 V=8.0
MOVL C02447 V=8.0
MOVL C02448 V=8.0
MOVL C02449 V=8.0
MOVJ C02450 VJ=0.78
MOVJ C02451 VJ=0.78
MOVL C02452 V=11.7
TIMER T=2.00
MOVL C02453 V=11.7
MOVJ C02454 VJ=0.78
MOVJ C02455 VJ=0.78
MOVL C02456 V=8.0
MOVL C02457 V=8.0
MOVL C02458 V=8.0
MOVL C02459 V=8.0
MOVL C02460 V=8.0
MOVL C02461 V=8.0
MOVL C02462 V=8.0
MOVL C02463 V=8.0
MOVL C02464 V=8.0
MOVL C02465 V=8.0
MOVL C02466 V=8.0
MOVL C02467 V=8.0
MOVL C02468 V=8.0
MOVL C02469 V=8.0
MOVL C02470 V=8.0
MOVL C02471 V=8.0
MOVL C02472 V=8.0
MOVL C02473 V=8.0
MOVL C02474 V=8.0
MOVL C02475 V=8.0
MOVL C02476 V=8.0
MOVL C02477 V=8.0
MOVL C02478 V=8.0
MOVL C02479 V=8.0
MOVL C02480 V=8.0
MOVL C02481 V=8.0
MOVL C02482 V=8.0
MOVL C02483 V=8.0
MOVL C02484 V=8.0
MOVL C02485 V=8.0
MOVL C02486 V=8.0
MOVL C02487 V=8.0
MOVL C02488 V=8.0
MOVL C02489 V=8.0
MOVL C02490 V=8.0
MOVL C02491 V=8.0
MOVL C02492 V=8.0
MOVL C02493 V=8.0
MOVL C02494 V=8.0
MOVL C02495 V=8.0
MOVL C02496 V=8.0
MOVL C02497 V=8.0
MOVJ C02498 VJ=0.78
MOVL C02499 V=8.0
MOVL C02500 V=8.0
MOVL C02501 V=8.0
MOVL C02502 V=8.0
MOVL C02503 V=8.0
MOVL C02504 V=8.0
MOVL C02505 V=8.0
MOVL C02506 V=8.0
MOVL C02507 V=8.0
MOVL C02508 V=8.0
MOVL C02509 V=8.0
MOVL C02510 V=8.0
MOVL C02511 V=8.0
MOVL C02512 V=8.0
MOVL C02513 V=8.0
MOVL C02514 V=8.0
MOVL C02515 V=8.0
MOVL C02516 V=8.0
MOVL C02517 V=8.0
MOVL C02518 V=8.0
MOVL C02519 V=8.0
MOVL C02520 V=8.0
MOVL C02521 V=8.0
MOVL C02522 V=8.0
MOVL C02523 V=8.0
MOVL C02524 V=8.0
MOVL C02525 V=8.0
MOVL C02526 V=8.0
MOVL C02527 V=8.0
MOVL C02528 V=8.0
MOVL C02529 V=8.0
MOVL C02530 V=8.0
MOVL C02531 V=8.0
MOVL C02532 V=8.0
MOVL C02533 V=8.0
MOVL C02534 V=8.0
MOVL C02535 V=8.0
MOVL C02536 V=8.0
MOVL C02537 V=8.0
MOVL C02538 V=8.0
MOVL C02539 V=8.0
MOVL C02540 V=8.0
MOVL C02541 V=8.0
MOVL C02542 V=8.0
MOVL C02543 V=8.0
MOVL C02544 V=8.0
MOVL C02545 V=8.0
MOVL C02546 V=8.0
MOVL C02547 V=8.0
MOVL C02548 V=8.0
MOVL C02549 V=8.0
MOVL C02550 V=8.0
MOVL C02551 V=8.0
MOVL C02552 V=8.0
MOVL C02553 V=8.0
MOVL C02554 V=8.0
MOVL C02555 V=8.0
MOVL C02556 V=8.0
MOVL C02557 V=8.0
MOVL C02558 V=8.0
MOVL C02559 V=8.0
MOVL C02560 V=8.0
MOVJ C02561 VJ=0.78
MOVL C02562 V=8.0
MOVL C02563 V=8.0
MOVL C02564 V=8.0
MOVL C02565 V=8.0
MOVL C02566 V=8.0
MOVL C02567 V=8.0
MOVL C02568 V=8.0
MOVL C02569 V=8.0
MOVL C02570 V=8.0
MOVL C02571 V=8.0
MOVL C02572 V=8.0
MOVL C02573 V=8.0
MOVL C02574 V=8.0
MOVL C02575 V=8.0
MOVL C02576 V=8.0
MOVL C02577 V=8.0
MOVL C02578 V=8.0
MOVL C02579 V=8.0
MOVL C02580 V=8.0
MOVL C02581 V=8.0
MOVL C02582 V=8.0
MOVL C02583 V=8.0
MOVL C02584 V=8.0
MOVL C02585 V=8.0
MOVL C02586 V=8.0
MOVL C02587 V=8.0
MOVL C02588 V=8.0
MOVL C02589 V=8.0
MOVL C02590 V=8.0
MOVL C02591 V=8.0
MOVL C02592 V=8.0
MOVL C02593 V=8.0
MOVL C02594 V=8.0
MOVL C02595 V=8.0
MOVL C02596 V=8.0
MOVL C02597 V=8.0
MOVL C02598 V=8.0
MOVL C02599 V=8.0
MOVL C02600 V=8.0
MOVL C02601 V=8.0
MOVL C02602 V=8.0
MOVL C02603 V=8.0
MOVL C02604 V=8.0
MOVL C02605 V=8.0
MOVL C02606 V=8.0
MOVL C02607 V=8.0
MOVL C02608 V=8.0
MOVL C02609 V=8.0
MOVL C02610 V=8.0
MOVL C02611 V=8.0
MOVL C02612 V=8.0
MOVL C02613 V=8.0
MOVL C02614 V=8.0
MOVL C02615 V=8.0
MOVL C02616 V=8.0
MOVL C02617 V=8.0
MOVL C02618 V=8.0
MOVL C02619 V=8.0
MOVL C02620 V=8.0
MOVL C02621 V=8.0
MOVL C02622 V=8.0
MOVJ C02623 VJ=0.78
MOVJ C02624 VJ=0.78
MOVL C02625 V=11.7
TIMER T=2.00
MOVL C02626 V=11.7
MOVJ C02627 VJ=0.78
MOVJ C02628 VJ=0.78
MOVL C02629 V=8.0
MOVL C02630 V=8.0
MOVJ C02631 VJ=0.78
MOVL C02632 V=8.0
MOVL C02633 V=8.0
MOVL C02634 V=8.0
MOVL C02635 V=8.0
MOVL C02636 V=8.0
MOVL C02637 V=8.0
MOVL C02638 V=8.0
MOVL C02639 V=8.0
MOVL C02640 V=8.0
MOVL C02641 V=8.0
MOVL C02642 V=8.0
MOVL C02643 V=8.0
MOVL C02644 V=8.0
MOVL C02645 V=8.0
MOVL C02646 V=8.0
MOVL C02647 V=8.0
MOVL C02648 V=8.0
MOVL C02649 V=8.0
MOVL C02650 V=8.0
MOVL C02651 V=8.0
MOVL C02652 V=8.0
MOVL C02653 V=8.0
MOVL C02654 V=8.0
MOVL C02655 V=8.0
MOVL C02656 V=8.0
MOVL C02657 V=8.0
MOVL C02658 V=8.0
MOVL C02659 V=8.0
MOVL C02660 V=8.0
MOVL C02661 V=8.0
MOVL C02662 V=8.0
MOVL C02663 V=8.0
MOVL C02664 V=8.0
MOVL C02665 V=8.0
MOVL C02666 V=8.0
MOVL C02667 V=8.0
MOVL C02668 V=8.0
MOVL C02669 V=8.0
MOVL C02670 V=8.0
MOVL C02671 V=8.0
MOVL C02672 V=8.0
MOVL C02673 V=8.0
MOVL C02674 V=8.0
MOVL C02675 V=8.0
MOVL C02676 V=8.0
MOVL C02677 V=8.0
MOVL C02678 V=8.0
MOVL C02679 V=8.0
MOVL C02680 V=8.0
MOVL C02681 V=8.0
MOVL C02682 V=8.0
MOVL C02683 V=8.0
MOVL C02684 V=8.0
MOVL C02685 V=8.0
MOVL C02686 V=8.0
MOVL C02687 V=8.0
MOVL C02688 V=8.0
MOVL C02689 V=8.0
MOVL C02690 V=8.0
MOVL C02691 V=8.0
MOVL C02692 V=8.0
MOVL C02693 V=8.0
MOVJ C02694 VJ=0.78
MOVL C02695 V=8.0
MOVL C02696 V=8.0
MOVL C02697 V=8.0
MOVL C02698 V=8.0
MOVL C02699 V=8.0
MOVL C02700 V=8.0
MOVL C02701 V=8.0
MOVL C02702 V=8.0
MOVL C02703 V=8.0
MOVL C02704 V=8.0
MOVL C02705 V=8.0
MOVL C02706 V=8.0
MOVL C02707 V=8.0
MOVL C02708 V=8.0
MOVL C02709 V=8.0
MOVL C02710 V=8.0
MOVL C02711 V=8.0
MOVL C02712 V=8.0
MOVL C02713 V=8.0
MOVL C02714 V=8.0
MOVL C02715 V=8.0
MOVL C02716 V=8.0
MOVL C02717 V=8.0
MOVL C02718 V=8.0
MOVL C02719 V=8.0
MOVL C02720 V=8.0
MOVL C02721 V=8.0
MOVL C02722 V=8.0
MOVL C02723 V=8.0
MOVL C02724 V=8.0
MOVL C02725 V=8.0
MOVL C02726 V=8.0
MOVL C02727 V=8.0
MOVL C02728 V=8.0
MOVL C02729 V=8.0
MOVL C02730 V=8.0
MOVL C02731 V=8.0
MOVL C02732 V=8.0
MOVL C02733 V=8.0
MOVL C02734 V=8.0
MOVL C02735 V=8.0
MOVL C02736 V=8.0
MOVL C02737 V=8.0
MOVL C02738 V=8.0
MOVL C02739 V=8.0
MOVL C02740 V=8.0
MOVL C02741 V=8.0
MOVL C02742 V=8.0
MOVL C02743 V=8.0
MOVL C02744 V=8.0
MOVL C02745 V=8.0
MOVL C02746 V=8.0
MOVL C02747 V=8.0
MOVL C02748 V=8.0
MOVL C02749 V=8.0
MOVL C02750 V=8.0
MOVL C02751 V=8.0
MOVL C02752 V=8.0
MOVL C02753 V=8.0
MOVL C02754 V=8.0
MOVL C02755 V=8.0
MOVL C02756 V=8.0
MOVJ C02757 VJ=0.78
MOVL C02758 V=8.0
MOVL C02759 V=8.0
MOVL C02760 V=8.0
MOVL C02761 V=8.0
MOVL C02762 V=8.0
MOVL C02763 V=8.0
MOVL C02764 V=8.0
MOVL C02765 V=8.0
MOVL C02766 V=8.0
MOVL C02767 V=8.0
MOVL C02768 V=8.0
MOVL C02769 V=8.0
MOVL C02770 V=8.0
MOVL C02771 V=8.0
MOVL C02772 V=8.0
MOVL C02773 V=8.0
MOVL C02774 V=8.0
MOVL C02775 V=8.0
MOVL C02776 V=8.0
MOVL C02777 V=8.0
MOVL C02778 V=8.0
MOVL C02779 V=8.0
MOVL C02780 V=8.0
MOVL C02781 V=8.0
MOVL C02782 V=8.0
MOVL C02783 V=8.0
MOVL C02784 V=8.0
MOVL C02785 V=8.0
MOVL C02786 V=8.0
MOVL C02787 V=8.0
MOVL C02788 V=8.0
MOVL C02789 V=8.0
MOVL C02790 V=8.0
MOVL C02791 V=8.0
MOVL C02792 V=8.0
MOVL C02793 V=8.0
MOVL C02794 V=8.0
MOVL C02795 V=8.0
MOVL C02796 V=8.0
MOVL C02797 V=8.0
MOVL C02798 V=8.0
MOVJ C02799 VJ=0.78
MOVJ C02800 VJ=0.78
MOVL C02801 V=11.7
TIMER T=2.00
MOVL C02802 V=11.7
MOVJ C02803 VJ=0.78
MOVJ C02804 VJ=0.78
MOVL C02805 V=8.0
MOVL C02806 V=8.0
MOVL C02807 V=8.0
MOVL C02808 V=8.0
MOVL C02809 V=8.0
MOVL C02810 V=8.0
MOVL C02811 V=8.0
MOVL C02812 V=8.0
MOVL C02813 V=8.0
MOVL C02814 V=8.0
MOVL C02815 V=8.0
MOVL C02816 V=8.0
MOVL C02817 V=8.0
MOVL C02818 V=8.0
MOVL C02819 V=8.0
MOVL C02820 V=8.0
MOVL C02821 V=8.0
MOVL C02822 V=8.0
MOVL C02823 V=8.0
MOVL C02824 V=8.0
MOVL C02825 V=8.0
MOVL C02826 V=8.0
MOVJ C02827 VJ=0.78
MOVL C02828 V=8.0
MOVL C02829 V=8.0
MOVL C02830 V=8.0
MOVL C02831 V=8.0
MOVL C02832 V=8.0
MOVL C02833 V=8.0
MOVL C02834 V=8.0
MOVL C02835 V=8.0
MOVL C02836 V=8.0
MOVL C02837 V=8.0
MOVL C02838 V=8.0
MOVL C02839 V=8.0
MOVL C02840 V=8.0
MOVL C02841 V=8.0
MOVL C02842 V=8.0
MOVL C02843 V=8.0
MOVL C02844 V=8.0
MOVL C02845 V=8.0
MOVL C02846 V=8.0
MOVL C02847 V=8.0
MOVL C02848 V=8.0
MOVL C02849 V=8.0
MOVL C02850 V=8.0
MOVL C02851 V=8.0
MOVL C02852 V=8.0
MOVL C02853 V=8.0
MOVL C02854 V=8.0
MOVL C02855 V=8.0
MOVL C02856 V=8.0
MOVL C02857 V=8.0
MOVL C02858 V=8.0
MOVL C02859 V=8.0
MOVL C02860 V=8.0
MOVL C02861 V=8.0
MOVL C02862 V=8.0
MOVL C02863 V=8.0
MOVL C02864 V=8.0
MOVL C02865 V=8.0
MOVL C02866 V=8.0
MOVL C02867 V=8.0
MOVL C02868 V=8.0
MOVL C02869 V=8.0
MOVL C02870 V=8.0
MOVL C02871 V=8.0
MOVL C02872 V=8.0
MOVL C02873 V=8.0
MOVL C02874 V=8.0
MOVL C02875 V=8.0
MOVL C02876 V=8.0
MOVL C02877 V=8.0
MOVL C02878 V=8.0
MOVL C02879 V=8.0
MOVL C02880 V=8.0
MOVL C02881 V=8.0
MOVL C02882 V=8.0
MOVL C02883 V=8.0
MOVL C02884 V=8.0
MOVL C02885 V=8.0
MOVL C02886 V=8.0
MOVL C02887 V=8.0
MOVL C02888 V=8.0
MOVL C02889 V=8.0
MOVJ C02890 VJ=0.78
MOVL C02891 V=8.0
MOVL C02892 V=8.0
MOVL C02893 V=8.0
MOVL C02894 V=8.0
MOVL C02895 V=8.0
MOVL C02896 V=8.0
MOVL C02897 V=8.0
MOVL C02898 V=8.0
MOVL C02899 V=8.0
MOVL C02900 V=8.0
MOVL C02901 V=8.0
MOVL C02902 V=8.0
MOVL C02903 V=8.0
MOVL C02904 V=8.0
MOVL C02905 V=8.0
MOVL C02906 V=8.0
MOVL C02907 V=8.0
MOVL C02908 V=8.0
MOVL C02909 V=8.0
MOVL C02910 V=8.0
MOVL C02911 V=8.0
MOVL C02912 V=8.0
MOVL C02913 V=8.0
MOVL C02914 V=8.0
MOVL C02915 V=8.0
MOVL C02916 V=8.0
MOVL C02917 V=8.0
MOVL C02918 V=8.0
MOVL C02919 V=8.0
MOVL C02920 V=8.0
MOVL C02921 V=8.0
MOVL C02922 V=8.0
MOVL C02923 V=8.0
MOVL C02924 V=8.0
MOVL C02925 V=8.0
MOVL C02926 V=8.0
MOVL C02927 V=8.0
MOVL C02928 V=8.0
MOVL C02929 V=8.0
MOVL C02930 V=8.0
MOVL C02931 V=8.0
MOVL C02932 V=8.0
MOVL C02933 V=8.0
MOVL C02934 V=8.0
MOVL C02935 V=8.0
MOVL C02936 V=8.0
MOVL C02937 V=8.0
MOVL C02938 V=8.0
MOVL C02939 V=8.0
MOVL C02940 V=8.0
MOVL C02941 V=8.0
MOVL C02942 V=8.0
MOVL C02943 V=8.0
MOVL C02944 V=8.0
MOVL C02945 V=8.0
MOVL C02946 V=8.0
MOVL C02947 V=8.0
MOVL C02948 V=8.0
MOVL C02949 V=8.0
MOVL C02950 V=8.0
MOVL C02951 V=8.0
MOVL C02952 V=8.0
MOVJ C02953 VJ=0.78
MOVL C02954 V=8.0
MOVL C02955 V=8.0
MOVL C02956 V=8.0
MOVL C02957 V=8.0
MOVL C02958 V=8.0
MOVL C02959 V=8.0
MOVL C02960 V=8.0
MOVL C02961 V=8.0
MOVL C02962 V=8.0
MOVL C02963 V=8.0
MOVL C02964 V=8.0
MOVL C02965 V=8.0
MOVL C02966 V=8.0
MOVL C02967 V=8.0
MOVL C02968 V=8.0
MOVL C02969 V=8.0
MOVL C02970 V=8.0
MOVL C02971 V=8.0
MOVL C02972 V=8.0
MOVL C02973 V=8.0
MOVL C02974 V=8.0
MOVJ C02975 VJ=0.78
MOVJ C02976 VJ=0.78
MOVL C02977 V=11.7
TIMER T=2.00
MOVL C02978 V=11.7
MOVJ C02979 VJ=0.78
MOVJ C02980 VJ=0.78
MOVL C02981 V=8.0
MOVL C02982 V=8.0
MOVL C02983 V=8.0
MOVL C02984 V=8.0
MOVL C02985 V=8.0
MOVL C02986 V=8.0
MOVL C02987 V=8.0
MOVL C02988 V=8.0
MOVL C02989 V=8.0
MOVL C02990 V=8.0
MOVL C02991 V=8.0
MOVL C02992 V=8.0
MOVL C02993 V=8.0
MOVL C02994 V=8.0
MOVL C02995 V=8.0
MOVL C02996 V=8.0
MOVL C02997 V=8.0
MOVL C02998 V=8.0
MOVL C02999 V=8.0
MOVL C03000 V=8.0
MOVL C03001 V=8.0
MOVL C03002 V=8.0
MOVL C03003 V=8.0
MOVL C03004 V=8.0
MOVL C03005 V=8.0
MOVL C03006 V=8.0
MOVL C03007 V=8.0
MOVL C03008 V=8.0
MOVL C03009 V=8.0
MOVL C03010 V=8.0
MOVL C03011 V=8.0
MOVL C03012 V=8.0
MOVL C03013 V=8.0
MOVL C03014 V=8.0
MOVL C03015 V=8.0
MOVL C03016 V=8.0
MOVL C03017 V=8.0
MOVL C03018 V=8.0
MOVL C03019 V=8.0
MOVL C03020 V=8.0
MOVL C03021 V=8.0
MOVL C03022 V=8.0
MOVJ C03023 VJ=0.78
MOVL C03024 V=8.0
MOVL C03025 V=8.0
MOVL C03026 V=8.0
MOVL C03027 V=8.0
MOVL C03028 V=8.0
MOVL C03029 V=8.0
MOVL C03030 V=8.0
MOVL C03031 V=8.0
MOVL C03032 V=8.0
MOVL C03033 V=8.0
MOVL C03034 V=8.0
MOVL C03035 V=8.0
MOVL C03036 V=8.0
MOVL C03037 V=8.0
MOVL C03038 V=8.0
MOVL C03039 V=8.0
MOVL C03040 V=8.0
MOVL C03041 V=8.0
MOVL C03042 V=8.0
MOVL C03043 V=8.0
MOVL C03044 V=8.0
MOVL C03045 V=8.0
MOVL C03046 V=8.0
MOVL C03047 V=8.0
MOVL C03048 V=8.0
MOVL C03049 V=8.0
MOVL C03050 V=8.0
MOVL C03051 V=8.0
MOVL C03052 V=8.0
MOVL C03053 V=8.0
MOVL C03054 V=8.0
MOVL C03055 V=8.0
MOVL C03056 V=8.0
MOVL C03057 V=8.0
MOVL C03058 V=8.0
MOVL C03059 V=8.0
MOVL C03060 V=8.0
MOVL C03061 V=8.0
MOVL C03062 V=8.0
MOVL C03063 V=8.0
MOVL C03064 V=8.0
MOVL C03065 V=8.0
MOVL C03066 V=8.0
MOVL C03067 V=8.0
MOVL C03068 V=8.0
MOVL C03069 V=8.0
MOVL C03070 V=8.0
MOVL C03071 V=8.0
MOVL C03072 V=8.0
MOVL C03073 V=8.0
MOVL C03074 V=8.0
MOVL C03075 V=8.0
MOVL C03076 V=8.0
MOVL C03077 V=8.0
MOVL C03078 V=8.0
MOVL C03079 V=8.0
MOVL C03080 V=8.0
MOVL C03081 V=8.0
MOVL C03082 V=8.0
MOVL C03083 V=8.0
MOVL C03084 V=8.0
MOVL C03085 V=8.0
MOVJ C03086 VJ=0.78
MOVL C03087 V=8.0
MOVL C03088 V=8.0
MOVL C03089 V=8.0
MOVL C03090 V=8.0
MOVL C03091 V=8.0
MOVL C03092 V=8.0
MOVL C03093 V=8.0
MOVL C03094 V=8.0
MOVL C03095 V=8.0
MOVL C03096 V=8.0
MOVL C03097 V=8.0
MOVL C03098 V=8.0
MOVL C03099 V=8.0
MOVL C03100 V=8.0
MOVL C03101 V=8.0
MOVL C03102 V=8.0
MOVL C03103 V=8.0
MOVL C03104 V=8.0
MOVL C03105 V=8.0
MOVL C03106 V=8.0
MOVL C03107 V=8.0
MOVL C03108 V=8.0
MOVL C03109 V=8.0
MOVL C03110 V=8.0
MOVL C03111 V=8.0
MOVL C03112 V=8.0
MOVL C03113 V=8.0
MOVL C03114 V=8.0
MOVL C03115 V=8.0
MOVL C03116 V=8.0
MOVL C03117 V=8.0
MOVL C03118 V=8.0
MOVL C03119 V=8.0
MOVL C03120 V=8.0
MOVL C03121 V=8.0
MOVL C03122 V=8.0
MOVL C03123 V=8.0
MOVL C03124 V=8.0
MOVL C03125 V=8.0
MOVL C03126 V=8.0
MOVL C03127 V=8.0
MOVL C03128 V=8.0
MOVL C03129 V=8.0
MOVL C03130 V=8.0
MOVL C03131 V=8.0
MOVL C03132 V=8.0
MOVL C03133 V=8.0
MOVL C03134 V=8.0
MOVL C03135 V=8.0
MOVL C03136 V=8.0
MOVL C03137 V=8.0
MOVL C03138 V=8.0
MOVL C03139 V=8.0
MOVL C03140 V=8.0
MOVL C03141 V=8.0
MOVL C03142 V=8.0
MOVL C03143 V=8.0
MOVL C03144 V=8.0
MOVL C03145 V=8.0
MOVL C03146 V=8.0
MOVL C03147 V=8.0
MOVJ C03148 VJ=0.78
MOVJ C03149 VJ=0.78
MOVL C03150 V=11.7
TIMER T=2.00
MOVL C03151 V=11.7
MOVJ C03152 VJ=0.78
MOVJ C03153 VJ=0.78
MOVL C03154 V=8.0
MOVL C03155 V=8.0
MOVJ C03156 VJ=0.78
MOVL C03157 V=8.0
MOVL C03158 V=8.0
MOVL C03159 V=8.0
MOVL C03160 V=8.0
MOVL C03161 V=8.0
MOVL C03162 V=8.0
MOVL C03163 V=8.0
MOVL C03164 V=8.0
MOVL C03165 V=8.0
MOVL C03166 V=8.0
MOVL C03167 V=8.0
MOVL C03168 V=8.0
MOVL C03169 V=8.0
MOVL C03170 V=8.0
MOVL C03171 V=8.0
MOVL C03172 V=8.0
MOVL C03173 V=8.0
MOVL C03174 V=8.0
MOVL C03175 V=8.0
MOVL C03176 V=8.0
MOVL C03177 V=8.0
MOVL C03178 V=8.0
MOVL C03179 V=8.0
MOVL C03180 V=8.0
MOVL C03181 V=8.0
MOVL C03182 V=8.0
MOVL C03183 V=8.0
MOVL C03184 V=8.0
MOVL C03185 V=8.0
MOVL C03186 V=8.0
MOVL C03187 V=8.0
MOVL C03188 V=8.0
MOVL C03189 V=8.0
MOVL C03190 V=8.0
MOVL C03191 V=8.0
MOVL C03192 V=8.0
MOVL C03193 V=8.0
MOVL C03194 V=8.0
MOVL C03195 V=8.0
MOVL C03196 V=8.0
MOVL C03197 V=8.0
MOVL C03198 V=8.0
MOVL C03199 V=8.0
MOVL C03200 V=8.0
MOVL C03201 V=8.0
MOVL C03202 V=8.0
MOVL C03203 V=8.0
MOVL C03204 V=8.0
MOVL C03205 V=8.0
MOVL C03206 V=8.0
MOVL C03207 V=8.0
MOVL C03208 V=8.0
MOVL C03209 V=8.0
MOVL C03210 V=8.0
MOVL C03211 V=8.0
MOVL C03212 V=8.0
MOVL C03213 V=8.0
MOVL C03214 V=8.0
MOVL C03215 V=8.0
MOVL C03216 V=8.0
MOVL C03217 V=8.0
MOVL C03218 V=8.0
MOVJ C03219 VJ=0.78
MOVL C03220 V=8.0
MOVL C03221 V=8.0
MOVL C03222 V=8.0
MOVL C03223 V=8.0
MOVL C03224 V=8.0
MOVL C03225 V=8.0
MOVL C03226 V=8.0
MOVL C03227 V=8.0
MOVL C03228 V=8.0
MOVL C03229 V=8.0
MOVL C03230 V=8.0
MOVL C03231 V=8.0
MOVL C03232 V=8.0
MOVL C03233 V=8.0
MOVL C03234 V=8.0
MOVL C03235 V=8.0
MOVL C03236 V=8.0
MOVL C03237 V=8.0
MOVL C03238 V=8.0
MOVL C03239 V=8.0
MOVL C03240 V=8.0
MOVL C03241 V=8.0
MOVL C03242 V=8.0
MOVL C03243 V=8.0
MOVL C03244 V=8.0
MOVL C03245 V=8.0
MOVL C03246 V=8.0
MOVL C03247 V=8.0
MOVL C03248 V=8.0
MOVL C03249 V=8.0
MOVL C03250 V=8.0
MOVL C03251 V=8.0
MOVL C03252 V=8.0
MOVL C03253 V=8.0
MOVL C03254 V=8.0
MOVL C03255 V=8.0
MOVL C03256 V=8.0
MOVL C03257 V=8.0
MOVL C03258 V=8.0
MOVL C03259 V=8.0
MOVL C03260 V=8.0
MOVL C03261 V=8.0
MOVL C03262 V=8.0
MOVL C03263 V=8.0
MOVL C03264 V=8.0
MOVL C03265 V=8.0
MOVL C03266 V=8.0
MOVL C03267 V=8.0
MOVL C03268 V=8.0
MOVL C03269 V=8.0
MOVL C03270 V=8.0
MOVL C03271 V=8.0
MOVL C03272 V=8.0
MOVL C03273 V=8.0
MOVL C03274 V=8.0
MOVL C03275 V=8.0
MOVL C03276 V=8.0
MOVL C03277 V=8.0
MOVL C03278 V=8.0
MOVL C03279 V=8.0
MOVL C03280 V=8.0
MOVL C03281 V=8.0
MOVJ C03282 VJ=0.78
MOVL C03283 V=8.0
MOVL C03284 V=8.0
MOVL C03285 V=8.0
MOVL C03286 V=8.0
MOVL C03287 V=8.0
MOVL C03288 V=8.0
MOVL C03289 V=8.0
MOVL C03290 V=8.0
MOVL C03291 V=8.0
MOVL C03292 V=8.0
MOVL C03293 V=8.0
MOVL C03294 V=8.0
MOVL C03295 V=8.0
MOVL C03296 V=8.0
MOVL C03297 V=8.0
MOVL C03298 V=8.0
MOVL C03299 V=8.0
MOVL C03300 V=8.0
MOVL C03301 V=8.0
MOVL C03302 V=8.0
MOVL C03303 V=8.0
MOVL C03304 V=8.0
MOVL C03305 V=8.0
MOVL C03306 V=8.0
MOVL C03307 V=8.0
MOVL C03308 V=8.0
MOVL C03309 V=8.0
MOVL C03310 V=8.0
MOVL C03311 V=8.0
MOVL C03312 V=8.0
MOVL C03313 V=8.0
MOVL C03314 V=8.0
MOVL C03315 V=8.0
MOVL C03316 V=8.0
MOVL C03317 V=8.0
MOVL C03318 V=8.0
MOVL C03319 V=8.0
MOVL C03320 V=8.0
MOVL C03321 V=8.0
MOVL C03322 V=8.0
MOVL C03323 V=8.0
MOVJ C03324 VJ=0.78
MOVJ C03325 VJ=0.78
MOVL C03326 V=11.7
TIMER T=2.00
MOVL C03327 V=11.7
MOVJ C03328 VJ=0.78
MOVJ C03329 VJ=0.78
MOVL C03330 V=8.0
MOVL C03331 V=8.0
MOVL C03332 V=8.0
MOVL C03333 V=8.0
MOVL C03334 V=8.0
MOVL C03335 V=8.0
MOVL C03336 V=8.0
MOVL C03337 V=8.0
MOVL C03338 V=8.0
MOVL C03339 V=8.0
MOVL C03340 V=8.0
MOVL C03341 V=8.0
MOVL C03342 V=8.0
MOVL C03343 V=8.0
MOVL C03344 V=8.0
MOVL C03345 V=8.0
MOVL C03346 V=8.0
MOVL C03347 V=8.0
MOVL C03348 V=8.0
MOVL C03349 V=8.0
MOVL C03350 V=8.0
MOVL C03351 V=8.0
MOVJ C03352 VJ=0.78
MOVL C03353 V=8.0
MOVL C03354 V=8.0
MOVL C03355 V=8.0
MOVL C03356 V=8.0
MOVL C03357 V=8.0
MOVL C03358 V=8.0
MOVL C03359 V=8.0
MOVL C03360 V=8.0
MOVL C03361 V=8.0
MOVL C03362 V=8.0
MOVL C03363 V=8.0
MOVL C03364 V=8.0
MOVL C03365 V=8.0
MOVL C03366 V=8.0
MOVL C03367 V=8.0
MOVL C03368 V=8.0
MOVL C03369 V=8.0
MOVL C03370 V=8.0
MOVL C03371 V=8.0
MOVL C03372 V=8.0
MOVL C03373 V=8.0
MOVL C03374 V=8.0
MOVL C03375 V=8.0
MOVL C03376 V=8.0
MOVL C03377 V=8.0
MOVL C03378 V=8.0
MOVL C03379 V=8.0
MOVL C03380 V=8.0
MOVL C03381 V=8.0
MOVL C03382 V=8.0
MOVL C03383 V=8.0
MOVL C03384 V=8.0
MOVL C03385 V=8.0
MOVL C03386 V=8.0
MOVL C03387 V=8.0
MOVL C03388 V=8.0
MOVL C03389 V=8.0
MOVL C03390 V=8.0
MOVL C03391 V=8.0
MOVL C03392 V=8.0
MOVL C03393 V=8.0
MOVL C03394 V=8.0
MOVL C03395 V=8.0
MOVL C03396 V=8.0
MOVL C03397 V=8.0
MOVL C03398 V=8.0
MOVL C03399 V=8.0
MOVL C03400 V=8.0
MOVL C03401 V=8.0
MOVL C03402 V=8.0
MOVL C03403 V=8.0
MOVL C03404 V=8.0
MOVL C03405 V=8.0
MOVL C03406 V=8.0
MOVL C03407 V=8.0
MOVL C03408 V=8.0
MOVL C03409 V=8.0
MOVL C03410 V=8.0
MOVL C03411 V=8.0
MOVL C03412 V=8.0
MOVL C03413 V=8.0
MOVL C03414 V=8.0
MOVJ C03415 VJ=0.78
MOVL C03416 V=8.0
MOVL C03417 V=8.0
MOVL C03418 V=8.0
MOVL C03419 V=8.0
MOVL C03420 V=8.0
MOVL C03421 V=8.0
MOVL C03422 V=8.0
MOVL C03423 V=8.0
MOVL C03424 V=8.0
MOVL C03425 V=8.0
MOVL C03426 V=8.0
MOVL C03427 V=8.0
MOVL C03428 V=8.0
MOVL C03429 V=8.0
MOVL C03430 V=8.0
MOVL C03431 V=8.0
MOVL C03432 V=8.0
MOVL C03433 V=8.0
MOVL C03434 V=8.0
MOVL C03435 V=8.0
MOVL C03436 V=8.0
MOVL C03437 V=8.0
MOVL C03438 V=8.0
MOVL C03439 V=8.0
MOVL C03440 V=8.0
MOVL C03441 V=8.0
MOVL C03442 V=8.0
MOVL C03443 V=8.0
MOVL C03444 V=8.0
MOVL C03445 V=8.0
MOVL C03446 V=8.0
MOVL C03447 V=8.0
MOVL C03448 V=8.0
MOVL C03449 V=8.0
MOVL C03450 V=8.0
MOVL C03451 V=8.0
MOVL C03452 V=8.0
MOVL C03453 V=8.0
MOVL C03454 V=8.0
MOVL C03455 V=8.0
MOVL C03456 V=8.0
MOVL C03457 V=8.0
MOVL C03458 V=8.0
MOVL C03459 V=8.0
MOVL C03460 V=8.0
MOVL C03461 V=8.0
MOVL C03462 V=8.0
MOVL C03463 V=8.0
MOVL C03464 V=8.0
MOVL C03465 V=8.0
MOVL C03466 V=8.0
MOVL C03467 V=8.0
MOVL C03468 V=8.0
MOVL C03469 V=8.0
MOVL C03470 V=8.0
MOVL C03471 V=8.0
MOVL C03472 V=8.0
MOVL C03473 V=8.0
MOVL C03474 V=8.0
MOVL C03475 V=8.0
MOVL C03476 V=8.0
MOVL C03477 V=8.0
MOVJ C03478 VJ=0.78
MOVL C03479 V=8.0
MOVL C03480 V=8.0
MOVL C03481 V=8.0
MOVL C03482 V=8.0
MOVL C03483 V=8.0
MOVL C03484 V=8.0
MOVL C03485 V=8.0
MOVL C03486 V=8.0
MOVL C03487 V=8.0
MOVL C03488 V=8.0
MOVL C03489 V=8.0
MOVL C03490 V=8.0
MOVL C03491 V=8.0
MOVL C03492 V=8.0
MOVL C03493 V=8.0
MOVL C03494 V=8.0
MOVL C03495 V=8.0
MOVL C03496 V=8.0
MOVL C03497 V=8.0
MOVL C03498 V=8.0
MOVL C03499 V=8.0
MOVJ C03500 VJ=0.78
MOVJ C03501 VJ=0.78
MOVL C03502 V=11.7
TIMER T=2.00
MOVL C03503 V=11.7
MOVJ C03504 VJ=0.78
MOVJ C03505 VJ=0.78
MOVL C03506 V=8.0
MOVL C03507 V=8.0
MOVL C03508 V=8.0
MOVL C03509 V=8.0
MOVL C03510 V=8.0
MOVL C03511 V=8.0
MOVL C03512 V=8.0
MOVL C03513 V=8.0
MOVL C03514 V=8.0
MOVL C03515 V=8.0
MOVL C03516 V=8.0
MOVL C03517 V=8.0
MOVL C03518 V=8.0
MOVL C03519 V=8.0
MOVL C03520 V=8.0
MOVL C03521 V=8.0
MOVL C03522 V=8.0
MOVL C03523 V=8.0
MOVL C03524 V=8.0
MOVL C03525 V=8.0
MOVL C03526 V=8.0
MOVL C03527 V=8.0
MOVL C03528 V=8.0
MOVL C03529 V=8.0
MOVL C03530 V=8.0
MOVL C03531 V=8.0
MOVL C03532 V=8.0
MOVL C03533 V=8.0
MOVL C03534 V=8.0
MOVL C03535 V=8.0
MOVL C03536 V=8.0
MOVL C03537 V=8.0
MOVL C03538 V=8.0
MOVL C03539 V=8.0
MOVL C03540 V=8.0
MOVL C03541 V=8.0
MOVL C03542 V=8.0
MOVL C03543 V=8.0
MOVL C03544 V=8.0
MOVL C03545 V=8.0
MOVL C03546 V=8.0
MOVL C03547 V=8.0
MOVJ C03548 VJ=0.78
MOVL C03549 V=8.0
MOVL C03550 V=8.0
MOVL C03551 V=8.0
MOVL C03552 V=8.0
MOVL C03553 V=8.0
MOVL C03554 V=8.0
MOVL C03555 V=8.0
MOVL C03556 V=8.0
MOVL C03557 V=8.0
MOVL C03558 V=8.0
MOVL C03559 V=8.0
MOVL C03560 V=8.0
MOVL C03561 V=8.0
MOVL C03562 V=8.0
MOVL C03563 V=8.0
MOVL C03564 V=8.0
MOVL C03565 V=8.0
MOVL C03566 V=8.0
MOVL C03567 V=8.0
MOVL C03568 V=8.0
MOVL C03569 V=8.0
MOVL C03570 V=8.0
MOVL C03571 V=8.0
MOVL C03572 V=8.0
MOVL C03573 V=8.0
MOVL C03574 V=8.0
MOVL C03575 V=8.0
MOVL C03576 V=8.0
MOVL C03577 V=8.0
MOVL C03578 V=8.0
MOVL C03579 V=8.0
MOVL C03580 V=8.0
MOVL C03581 V=8.0
MOVL C03582 V=8.0
MOVL C03583 V=8.0
MOVL C03584 V=8.0
MOVL C03585 V=8.0
MOVL C03586 V=8.0
MOVL C03587 V=8.0
MOVL C03588 V=8.0
MOVL C03589 V=8.0
MOVL C03590 V=8.0
MOVL C03591 V=8.0
MOVL C03592 V=8.0
MOVL C03593 V=8.0
MOVL C03594 V=8.0
MOVL C03595 V=8.0
MOVL C03596 V=8.0
MOVL C03597 V=8.0
MOVL C03598 V=8.0
MOVL C03599 V=8.0
MOVL C03600 V=8.0
MOVL C03601 V=8.0
MOVL C03602 V=8.0
MOVL C03603 V=8.0
MOVL C03604 V=8.0
MOVL C03605 V=8.0
MOVL C03606 V=8.0
MOVL C03607 V=8.0
MOVL C03608 V=8.0
MOVL C03609 V=8.0
MOVL C03610 V=8.0
MOVJ C03611 VJ=0.78
MOVL C03612 V=8.0
MOVL C03613 V=8.0
MOVL C03614 V=8.0
MOVL C03615 V=8.0
MOVL C03616 V=8.0
MOVL C03617 V=8.0
MOVL C03618 V=8.0
MOVL C03619 V=8.0
MOVL C03620 V=8.0
MOVL C03621 V=8.0
MOVL C03622 V=8.0
MOVL C03623 V=8.0
MOVL C03624 V=8.0
MOVL C03625 V=8.0
MOVL C03626 V=8.0
MOVL C03627 V=8.0
MOVL C03628 V=8.0
MOVL C03629 V=8.0
MOVL C03630 V=8.0
MOVL C03631 V=8.0
MOVL C03632 V=8.0
MOVL C03633 V=8.0
MOVL C03634 V=8.0
MOVL C03635 V=8.0
MOVL C03636 V=8.0
MOVL C03637 V=8.0
MOVL C03638 V=8.0
MOVL C03639 V=8.0
MOVL C03640 V=8.0
MOVL C03641 V=8.0
MOVL C03642 V=8.0
MOVL C03643 V=8.0
MOVL C03644 V=8.0
MOVL C03645 V=8.0
MOVL C03646 V=8.0
MOVL C03647 V=8.0
MOVL C03648 V=8.0
MOVL C03649 V=8.0
MOVL C03650 V=8.0
MOVL C03651 V=8.0
MOVL C03652 V=8.0
MOVL C03653 V=8.0
MOVL C03654 V=8.0
MOVL C03655 V=8.0
MOVL C03656 V=8.0
MOVL C03657 V=8.0
MOVL C03658 V=8.0
MOVL C03659 V=8.0
MOVL C03660 V=8.0
MOVL C03661 V=8.0
MOVL C03662 V=8.0
MOVL C03663 V=8.0
MOVL C03664 V=8.0
MOVL C03665 V=8.0
MOVL C03666 V=8.0
MOVL C03667 V=8.0
MOVL C03668 V=8.0
MOVL C03669 V=8.0
MOVL C03670 V=8.0
MOVL C03671 V=8.0
MOVL C03672 V=8.0
MOVJ C03673 VJ=0.78
MOVJ C03674 VJ=0.78
MOVL C03675 V=11.7
TIMER T=2.00
MOVL C03676 V=11.7
MOVJ C03677 VJ=0.78
MOVJ C03678 VJ=0.78
MOVL C03679 V=8.0
MOVL C03680 V=8.0
MOVJ C03681 VJ=0.78
MOVL C03682 V=8.0
MOVL C03683 V=8.0
MOVL C03684 V=8.0
MOVL C03685 V=8.0
MOVL C03686 V=8.0
MOVL C03687 V=8.0
MOVL C03688 V=8.0
MOVL C03689 V=8.0
MOVL C03690 V=8.0
MOVL C03691 V=8.0
MOVL C03692 V=8.0
MOVL C03693 V=8.0
MOVL C03694 V=8.0
MOVL C03695 V=8.0
MOVL C03696 V=8.0
MOVL C03697 V=8.0
MOVL C03698 V=8.0
MOVL C03699 V=8.0
MOVL C03700 V=8.0
MOVL C03701 V=8.0
MOVL C03702 V=8.0
MOVL C03703 V=8.0
MOVL C03704 V=8.0
MOVL C03705 V=8.0
MOVL C03706 V=8.0
MOVL C03707 V=8.0
MOVL C03708 V=8.0
MOVL C03709 V=8.0
MOVL C03710 V=8.0
MOVL C03711 V=8.0
MOVL C03712 V=8.0
MOVL C03713 V=8.0
MOVL C03714 V=8.0
MOVL C03715 V=8.0
MOVL C03716 V=8.0
MOVL C03717 V=8.0
MOVL C03718 V=8.0
MOVL C03719 V=8.0
MOVL C03720 V=8.0
MOVL C03721 V=8.0
MOVL C03722 V=8.0
MOVL C03723 V=8.0
MOVL C03724 V=8.0
MOVL C03725 V=8.0
MOVL C03726 V=8.0
MOVL C03727 V=8.0
MOVL C03728 V=8.0
MOVL C03729 V=8.0
MOVL C03730 V=8.0
MOVL C03731 V=8.0
MOVL C03732 V=8.0
MOVL C03733 V=8.0
MOVL C03734 V=8.0
MOVL C03735 V=8.0
MOVL C03736 V=8.0
MOVL C03737 V=8.0
MOVL C03738 V=8.0
MOVL C03739 V=8.0
MOVL C03740 V=8.0
MOVL C03741 V=8.0
MOVL C03742 V=8.0
MOVL C03743 V=8.0
MOVJ C03744 VJ=0.78
MOVL C03745 V=8.0
MOVL C03746 V=8.0
MOVL C03747 V=8.0
MOVL C03748 V=8.0
MOVL C03749 V=8.0
MOVL C03750 V=8.0
MOVL C03751 V=8.0
MOVL C03752 V=8.0
MOVL C03753 V=8.0
MOVL C03754 V=8.0
MOVL C03755 V=8.0
MOVL C03756 V=8.0
MOVL C03757 V=8.0
MOVL C03758 V=8.0
MOVL C03759 V=8.0
MOVL C03760 V=8.0
MOVL C03761 V=8.0
MOVL C03762 V=8.0
MOVL C03763 V=8.0
MOVL C03764 V=8.0
MOVL C03765 V=8.0
MOVL C03766 V=8.0
MOVL C03767 V=8.0
MOVL C03768 V=8.0
MOVL C03769 V=8.0
MOVL C03770 V=8.0
MOVL C03771 V=8.0
MOVL C03772 V=8.0
MOVL C03773 V=8.0
MOVL C03774 V=8.0
MOVL C03775 V=8.0
MOVL C03776 V=8.0
MOVL C03777 V=8.0
MOVL C03778 V=8.0
MOVL C03779 V=8.0
MOVL C03780 V=8.0
MOVL C03781 V=8.0
MOVL C03782 V=8.0
MOVL C03783 V=8.0
MOVL C03784 V=8.0
MOVL C03785 V=8.0
MOVL C03786 V=8.0
MOVL C03787 V=8.0
MOVL C03788 V=8.0
MOVL C03789 V=8.0
MOVL C03790 V=8.0
MOVL C03791 V=8.0
MOVL C03792 V=8.0
MOVL C03793 V=8.0
MOVL C03794 V=8.0
MOVL C03795 V=8.0
MOVL C03796 V=8.0
MOVL C03797 V=8.0
MOVL C03798 V=8.0
MOVL C03799 V=8.0
MOVL C03800 V=8.0
MOVL C03801 V=8.0
MOVL C03802 V=8.0
MOVL C03803 V=8.0
MOVL C03804 V=8.0
MOVL C03805 V=8.0
MOVL C03806 V=8.0
MOVJ C03807 VJ=0.78
MOVL C03808 V=8.0
MOVL C03809 V=8.0
MOVL C03810 V=8.0
MOVL C03811 V=8.0
MOVL C03812 V=8.0
MOVL C03813 V=8.0
MOVL C03814 V=8.0
MOVL C03815 V=8.0
MOVL C03816 V=8.0
MOVL C03817 V=8.0
MOVL C03818 V=8.0
MOVL C03819 V=8.0
MOVL C03820 V=8.0
MOVL C03821 V=8.0
MOVL C03822 V=8.0
MOVL C03823 V=8.0
MOVL C03824 V=8.0
MOVL C03825 V=8.0
MOVL C03826 V=8.0
MOVL C03827 V=8.0
MOVL C03828 V=8.0
MOVL C03829 V=8.0
MOVL C03830 V=8.0
MOVL C03831 V=8.0
MOVL C03832 V=8.0
MOVL C03833 V=8.0
MOVL C03834 V=8.0
MOVL C03835 V=8.0
MOVL C03836 V=8.0
MOVL C03837 V=8.0
MOVL C03838 V=8.0
MOVL C03839 V=8.0
MOVL C03840 V=8.0
MOVL C03841 V=8.0
MOVL C03842 V=8.0
MOVL C03843 V=8.0
MOVL C03844 V=8.0
MOVL C03845 V=8.0
MOVL C03846 V=8.0
MOVL C03847 V=8.0
MOVL C03848 V=8.0
MOVJ C03849 VJ=0.78
MOVJ C03850 VJ=0.78
MOVL C03851 V=11.7
TIMER T=2.00
MOVL C03852 V=11.7
MOVJ C03853 VJ=0.78
MOVJ C03854 VJ=0.78
MOVL C03855 V=8.0
MOVL C03856 V=8.0
MOVL C03857 V=8.0
MOVL C03858 V=8.0
MOVL C03859 V=8.0
MOVL C03860 V=8.0
MOVL C03861 V=8.0
MOVL C03862 V=8.0
MOVL C03863 V=8.0
MOVL C03864 V=8.0
MOVL C03865 V=8.0
MOVL C03866 V=8.0
MOVL C03867 V=8.0
MOVL C03868 V=8.0
MOVL C03869 V=8.0
MOVL C03870 V=8.0
MOVL C03871 V=8.0
MOVL C03872 V=8.0
MOVL C03873 V=8.0
MOVL C03874 V=8.0
MOVL C03875 V=8.0
MOVL C03876 V=8.0
MOVJ C03877 VJ=0.78
MOVL C03878 V=8.0
MOVL C03879 V=8.0
MOVL C03880 V=8.0
MOVL C03881 V=8.0
MOVL C03882 V=8.0
MOVL C03883 V=8.0
MOVL C03884 V=8.0
MOVL C03885 V=8.0
MOVL C03886 V=8.0
MOVL C03887 V=8.0
MOVL C03888 V=8.0
MOVL C03889 V=8.0
MOVL C03890 V=8.0
MOVL C03891 V=8.0
MOVL C03892 V=8.0
MOVL C03893 V=8.0
MOVL C03894 V=8.0
MOVL C03895 V=8.0
MOVL C03896 V=8.0
MOVL C03897 V=8.0
MOVL C03898 V=8.0
MOVL C03899 V=8.0
MOVL C03900 V=8.0
MOVL C03901 V=8.0
MOVL C03902 V=8.0
MOVL C03903 V=8.0
MOVL C03904 V=8.0
MOVL C03905 V=8.0
MOVL C03906 V=8.0
MOVL C03907 V=8.0
MOVL C03908 V=8.0
MOVL C03909 V=8.0
MOVL C03910 V=8.0
MOVL C03911 V=8.0
MOVL C03912 V=8.0
MOVL C03913 V=8.0
MOVL C03914 V=8.0
MOVL C03915 V=8.0
MOVL C03916 V=8.0
MOVL C03917 V=8.0
MOVL C03918 V=8.0
MOVL C03919 V=8.0
MOVL C03920 V=8.0
MOVL C03921 V=8.0
MOVL C03922 V=8.0
MOVL C03923 V=8.0
MOVL C03924 V=8.0
MOVL C03925 V=8.0
MOVL C03926 V=8.0
MOVL C03927 V=8.0
MOVL C03928 V=8.0
MOVL C03929 V=8.0
MOVL C03930 V=8.0
MOVL C03931 V=8.0
MOVL C03932 V=8.0
MOVL C03933 V=8.0
MOVL C03934 V=8.0
MOVL C03935 V=8.0
MOVL C03936 V=8.0
MOVL C03937 V=8.0
MOVL C03938 V=8.0
MOVL C03939 V=8.0
MOVJ C03940 VJ=0.78
MOVL C03941 V=8.0
MOVL C03942 V=8.0
MOVL C03943 V=8.0
MOVL C03944 V=8.0
MOVL C03945 V=8.0
MOVL C03946 V=8.0
MOVL C03947 V=8.0
MOVL C03948 V=8.0
MOVL C03949 V=8.0
MOVL C03950 V=8.0
MOVL C03951 V=8.0
MOVL C03952 V=8.0
MOVL C03953 V=8.0
MOVL C03954 V=8.0
MOVL C03955 V=8.0
MOVL C03956 V=8.0
MOVL C03957 V=8.0
MOVL C03958 V=8.0
MOVL C03959 V=8.0
MOVL C03960 V=8.0
MOVL C03961 V=8.0
MOVL C03962 V=8.0
MOVL C03963 V=8.0
MOVL C03964 V=8.0
MOVL C03965 V=8.0
MOVL C03966 V=8.0
MOVL C03967 V=8.0
MOVL C03968 V=8.0
MOVL C03969 V=8.0
MOVL C03970 V=8.0
MOVL C03971 V=8.0
MOVL C03972 V=8.0
MOVL C03973 V=8.0
MOVL C03974 V=8.0
MOVL C03975 V=8.0
MOVL C03976 V=8.0
MOVL C03977 V=8.0
MOVL C03978 V=8.0
MOVL C03979 V=8.0
MOVL C03980 V=8.0
MOVL C03981 V=8.0
MOVL C03982 V=8.0
MOVL C03983 V=8.0
MOVL C03984 V=8.0
MOVL C03985 V=8.0
MOVL C03986 V=8.0
MOVL C03987 V=8.0
MOVL C03988 V=8.0
MOVL C03989 V=8.0
MOVL C03990 V=8.0
MOVL C03991 V=8.0
MOVL C03992 V=8.0
MOVL C03993 V=8.0
MOVL C03994 V=8.0
MOVL C03995 V=8.0
MOVL C03996 V=8.0
MOVL C03997 V=8.0
MOVL C03998 V=8.0
MOVL C03999 V=8.0
MOVL C04000 V=8.0
MOVL C04001 V=8.0
MOVL C04002 V=8.0
MOVJ C04003 VJ=0.78
MOVL C04004 V=8.0
MOVL C04005 V=8.0
MOVL C04006 V=8.0
MOVL C04007 V=8.0
MOVL C04008 V=8.0
MOVL C04009 V=8.0
MOVL C04010 V=8.0
MOVL C04011 V=8.0
MOVL C04012 V=8.0
MOVL C04013 V=8.0
MOVL C04014 V=8.0
MOVL C04015 V=8.0
MOVL C04016 V=8.0
MOVL C04017 V=8.0
MOVL C04018 V=8.0
MOVL C04019 V=8.0
MOVL C04020 V=8.0
MOVL C04021 V=8.0
MOVL C04022 V=8.0
MOVL C04023 V=8.0
MOVL C04024 V=8.0
MOVJ C04025 VJ=0.78
MOVJ C04026 VJ=0.78
MOVL C04027 V=11.7
TIMER T=2.00
MOVL C04028 V=11.7
MOVJ C04029 VJ=0.78
MOVJ C04030 VJ=0.78
MOVL C04031 V=8.0
MOVL C04032 V=8.0
MOVL C04033 V=8.0
MOVL C04034 V=8.0
MOVL C04035 V=8.0
MOVL C04036 V=8.0
MOVL C04037 V=8.0
MOVL C04038 V=8.0
MOVL C04039 V=8.0
MOVL C04040 V=8.0
MOVL C04041 V=8.0
MOVL C04042 V=8.0
MOVL C04043 V=8.0
MOVL C04044 V=8.0
MOVL C04045 V=8.0
MOVL C04046 V=8.0
MOVL C04047 V=8.0
MOVL C04048 V=8.0
MOVL C04049 V=8.0
MOVL C04050 V=8.0
MOVL C04051 V=8.0
MOVL C04052 V=8.0
MOVL C04053 V=8.0
MOVL C04054 V=8.0
MOVL C04055 V=8.0
MOVL C04056 V=8.0
MOVL C04057 V=8.0
MOVL C04058 V=8.0
MOVL C04059 V=8.0
MOVL C04060 V=8.0
MOVL C04061 V=8.0
MOVL C04062 V=8.0
MOVL C04063 V=8.0
MOVL C04064 V=8.0
MOVL C04065 V=8.0
MOVL C04066 V=8.0
MOVL C04067 V=8.0
MOVL C04068 V=8.0
MOVL C04069 V=8.0
MOVL C04070 V=8.0
MOVL C04071 V=8.0
MOVL C04072 V=8.0
MOVJ C04073 VJ=0.78
MOVL C04074 V=8.0
MOVL C04075 V=8.0
MOVL C04076 V=8.0
MOVL C04077 V=8.0
MOVL C04078 V=8.0
MOVL C04079 V=8.0
MOVL C04080 V=8.0
MOVL C04081 V=8.0
MOVL C04082 V=8.0
MOVL C04083 V=8.0
MOVL C04084 V=8.0
MOVL C04085 V=8.0
MOVL C04086 V=8.0
MOVL C04087 V=8.0
MOVL C04088 V=8.0
MOVL C04089 V=8.0
MOVL C04090 V=8.0
MOVL C04091 V=8.0
MOVL C04092 V=8.0
MOVL C04093 V=8.0
MOVL C04094 V=8.0
MOVL C04095 V=8.0
MOVL C04096 V=8.0
MOVL C04097 V=8.0
MOVL C04098 V=8.0
MOVL C04099 V=8.0
MOVL C04100 V=8.0
MOVL C04101 V=8.0
MOVL C04102 V=8.0
MOVL C04103 V=8.0
MOVL C04104 V=8.0
MOVL C04105 V=8.0
MOVL C04106 V=8.0
MOVL C04107 V=8.0
MOVL C04108 V=8.0
MOVL C04109 V=8.0
MOVL C04110 V=8.0
MOVL C04111 V=8.0
MOVL C04112 V=8.0
MOVL C04113 V=8.0
MOVL C04114 V=8.0
MOVL C04115 V=8.0
MOVL C04116 V=8.0
MOVL C04117 V=8.0
MOVL C04118 V=8.0
MOVL C04119 V=8.0
MOVL C04120 V=8.0
MOVL C04121 V=8.0
MOVL C04122 V=8.0
MOVL C04123 V=8.0
MOVL C04124 V=8.0
MOVL C04125 V=8.0
MOVL C04126 V=8.0
MOVL C04127 V=8.0
MOVL C04128 V=8.0
MOVL C04129 V=8.0
MOVL C04130 V=8.0
MOVL C04131 V=8.0
MOVL C04132 V=8.0
MOVL C04133 V=8.0
MOVL C04134 V=8.0
MOVL C04135 V=8.0
MOVJ C04136 VJ=0.78
MOVL C04137 V=8.0
MOVL C04138 V=8.0
MOVL C04139 V=8.0
MOVL C04140 V=8.0
MOVL C04141 V=8.0
MOVL C04142 V=8.0
MOVL C04143 V=8.0
MOVL C04144 V=8.0
MOVL C04145 V=8.0
MOVL C04146 V=8.0
MOVL C04147 V=8.0
MOVL C04148 V=8.0
MOVL C04149 V=8.0
MOVL C04150 V=8.0
MOVL C04151 V=8.0
MOVL C04152 V=8.0
MOVL C04153 V=8.0
MOVL C04154 V=8.0
MOVL C04155 V=8.0
MOVL C04156 V=8.0
MOVL C04157 V=8.0
MOVL C04158 V=8.0
MOVL C04159 V=8.0
MOVL C04160 V=8.0
MOVL C04161 V=8.0
MOVL C04162 V=8.0
MOVL C04163 V=8.0
MOVL C04164 V=8.0
MOVL C04165 V=8.0
MOVL C04166 V=8.0
MOVL C04167 V=8.0
MOVL C04168 V=8.0
MOVL C04169 V=8.0
MOVL C04170 V=8.0
MOVL C04171 V=8.0
MOVL C04172 V=8.0
MOVL C04173 V=8.0
MOVL C04174 V=8.0
MOVL C04175 V=8.0
MOVL C04176 V=8.0
MOVL C04177 V=8.0
MOVL C04178 V=8.0
MOVL C04179 V=8.0
MOVL C04180 V=8.0
MOVL C04181 V=8.0
MOVL C04182 V=8.0
MOVL C04183 V=8.0
MOVL C04184 V=8.0
MOVL C04185 V=8.0
MOVL C04186 V=8.0
MOVL C04187 V=8.0
MOVL C04188 V=8.0
MOVL C04189 V=8.0
MOVL C04190 V=8.0
MOVL C04191 V=8.0
MOVL C04192 V=8.0
MOVL C04193 V=8.0
MOVL C04194 V=8.0
MOVL C04195 V=8.0
MOVL C04196 V=8.0
MOVL C04197 V=8.0
MOVJ C04198 VJ=0.78
MOVJ C04199 VJ=0.78
MOVL C04200 V=11.7
TIMER T=2.00
MOVL C04201 V=11.7
MOVJ C04202 VJ=0.78
MOVJ C04203 VJ=0.78
MOVL C04204 V=8.0
MOVL C04205 V=8.0
MOVJ C04206 VJ=0.78
MOVL C04207 V=8.0
MOVL C04208 V=8.0
MOVL C04209 V=8.0
MOVL C04210 V=8.0
MOVL C04211 V=8.0
MOVL C04212 V=8.0
MOVL C04213 V=8.0
MOVL C04214 V=8.0
MOVL C04215 V=8.0
MOVL C04216 V=8.0
MOVL C04217 V=8.0
MOVL C04218 V=8.0
MOVL C04219 V=8.0
MOVL C04220 V=8.0
MOVL C04221 V=8.0
MOVL C04222 V=8.0
MOVL C04223 V=8.0
MOVL C04224 V=8.0
MOVL C04225 V=8.0
MOVL C04226 V=8.0
MOVL C04227 V=8.0
MOVL C04228 V=8.0
MOVL C04229 V=8.0
MOVL C04230 V=8.0
MOVL C04231 V=8.0
MOVL C04232 V=8.0
MOVL C04233 V=8.0
MOVL C04234 V=8.0
MOVL C04235 V=8.0
MOVL C04236 V=8.0
MOVL C04237 V=8.0
MOVL C04238 V=8.0
MOVL C04239 V=8.0
MOVL C04240 V=8.0
MOVL C04241 V=8.0
MOVL C04242 V=8.0
MOVL C04243 V=8.0
MOVL C04244 V=8.0
MOVL C04245 V=8.0
MOVL C04246 V=8.0
MOVL C04247 V=8.0
MOVL C04248 V=8.0
MOVL C04249 V=8.0
MOVL C04250 V=8.0
MOVL C04251 V=8.0
MOVL C04252 V=8.0
MOVL C04253 V=8.0
MOVL C04254 V=8.0
MOVL C04255 V=8.0
MOVL C04256 V=8.0
MOVL C04257 V=8.0
MOVL C04258 V=8.0
MOVL C04259 V=8.0
MOVL C04260 V=8.0
MOVL C04261 V=8.0
MOVL C04262 V=8.0
MOVL C04263 V=8.0
MOVL C04264 V=8.0
MOVL C04265 V=8.0
MOVL C04266 V=8.0
MOVL C04267 V=8.0
MOVL C04268 V=8.0
MOVJ C04269 VJ=0.78
MOVL C04270 V=8.0
MOVL C04271 V=8.0
MOVL C04272 V=8.0
MOVL C04273 V=8.0
MOVL C04274 V=8.0
MOVL C04275 V=8.0
MOVL C04276 V=8.0
MOVL C04277 V=8.0
MOVL C04278 V=8.0
MOVL C04279 V=8.0
MOVL C04280 V=8.0
MOVL C04281 V=8.0
MOVL C04282 V=8.0
MOVL C04283 V=8.0
MOVL C04284 V=8.0
MOVL C04285 V=8.0
MOVL C04286 V=8.0
MOVL C04287 V=8.0
MOVL C04288 V=8.0
MOVL C04289 V=8.0
MOVL C04290 V=8.0
MOVL C04291 V=8.0
MOVL C04292 V=8.0
MOVL C04293 V=8.0
MOVL C04294 V=8.0
MOVL C04295 V=8.0
MOVL C04296 V=8.0
MOVL C04297 V=8.0
MOVL C04298 V=8.0
MOVL C04299 V=8.0
MOVL C04300 V=8.0
MOVL C04301 V=8.0
MOVL C04302 V=8.0
MOVL C04303 V=8.0
MOVL C04304 V=8.0
MOVL C04305 V=8.0
MOVL C04306 V=8.0
MOVL C04307 V=8.0
MOVL C04308 V=8.0
MOVL C04309 V=8.0
MOVL C04310 V=8.0
MOVL C04311 V=8.0
MOVL C04312 V=8.0
MOVL C04313 V=8.0
MOVL C04314 V=8.0
MOVL C04315 V=8.0
MOVL C04316 V=8.0
MOVL C04317 V=8.0
MOVL C04318 V=8.0
MOVL C04319 V=8.0
MOVL C04320 V=8.0
MOVL C04321 V=8.0
MOVL C04322 V=8.0
MOVL C04323 V=8.0
MOVL C04324 V=8.0
MOVL C04325 V=8.0
MOVL C04326 V=8.0
MOVL C04327 V=8.0
MOVL C04328 V=8.0
MOVL C04329 V=8.0
MOVL C04330 V=8.0
MOVL C04331 V=8.0
MOVJ C04332 VJ=0.78
MOVL C04333 V=8.0
MOVL C04334 V=8.0
MOVL C04335 V=8.0
MOVL C04336 V=8.0
MOVL C04337 V=8.0
MOVL C04338 V=8.0
MOVL C04339 V=8.0
MOVL C04340 V=8.0
MOVL C04341 V=8.0
MOVL C04342 V=8.0
MOVL C04343 V=8.0
MOVL C04344 V=8.0
MOVL C04345 V=8.0
MOVL C04346 V=8.0
MOVL C04347 V=8.0
MOVL C04348 V=8.0
MOVL C04349 V=8.0
MOVL C04350 V=8.0
MOVL C04351 V=8.0
MOVL C04352 V=8.0
MOVL C04353 V=8.0
MOVL C04354 V=8.0
MOVL C04355 V=8.0
MOVL C04356 V=8.0
MOVL C04357 V=8.0
MOVL C04358 V=8.0
MOVL C04359 V=8.0
MOVL C04360 V=8.0
MOVL C04361 V=8.0
MOVL C04362 V=8.0
MOVL C04363 V=8.0
MOVL C04364 V=8.0
MOVL C04365 V=8.0
MOVL C04366 V=8.0
MOVL C04367 V=8.0
MOVL C04368 V=8.0
MOVL C04369 V=8.0
MOVL C04370 V=8.0
MOVL C04371 V=8.0
MOVL C04372 V=8.0
MOVL C04373 V=8.0
MOVJ C04374 VJ=0.78
MOVJ C04375 VJ=0.78
MOVL C04376 V=11.7
TIMER T=2.00
MOVL C04377 V=11.7
MOVJ C04378 VJ=0.78
MOVJ C04379 VJ=0.78
MOVL C04380 V=8.0
MOVL C04381 V=8.0
MOVL C04382 V=8.0
MOVL C04383 V=8.0
MOVL C04384 V=8.0
MOVL C04385 V=8.0
MOVL C04386 V=8.0
MOVL C04387 V=8.0
MOVL C04388 V=8.0
MOVL C04389 V=8.0
MOVL C04390 V=8.0
MOVL C04391 V=8.0
MOVL C04392 V=8.0
MOVL C04393 V=8.0
MOVL C04394 V=8.0
MOVL C04395 V=8.0
MOVL C04396 V=8.0
MOVL C04397 V=8.0
MOVL C04398 V=8.0
MOVL C04399 V=8.0
MOVL C04400 V=8.0
MOVL C04401 V=8.0
MOVJ C04402 VJ=0.78
MOVL C04403 V=8.0
MOVL C04404 V=8.0
MOVL C04405 V=8.0
MOVL C04406 V=8.0
MOVL C04407 V=8.0
MOVL C04408 V=8.0
MOVL C04409 V=8.0
MOVL C04410 V=8.0
MOVL C04411 V=8.0
MOVL C04412 V=8.0
MOVL C04413 V=8.0
MOVL C04414 V=8.0
MOVL C04415 V=8.0
MOVL C04416 V=8.0
MOVL C04417 V=8.0
MOVL C04418 V=8.0
MOVL C04419 V=8.0
MOVL C04420 V=8.0
MOVL C04421 V=8.0
MOVL C04422 V=8.0
MOVL C04423 V=8.0
MOVL C04424 V=8.0
MOVL C04425 V=8.0
MOVL C04426 V=8.0
MOVL C04427 V=8.0
MOVL C04428 V=8.0
MOVL C04429 V=8.0
MOVL C04430 V=8.0
MOVL C04431 V=8.0
MOVL C04432 V=8.0
MOVL C04433 V=8.0
MOVL C04434 V=8.0
MOVL C04435 V=8.0
MOVL C04436 V=8.0
MOVL C04437 V=8.0
MOVL C04438 V=8.0
MOVL C04439 V=8.0
MOVL C04440 V=8.0
MOVL C04441 V=8.0
MOVL C04442 V=8.0
MOVL C04443 V=8.0
MOVL C04444 V=8.0
MOVL C04445 V=8.0
MOVL C04446 V=8.0
MOVL C04447 V=8.0
MOVL C04448 V=8.0
MOVL C04449 V=8.0
MOVL C04450 V=8.0
MOVL C04451 V=8.0
MOVL C04452 V=8.0
MOVL C04453 V=8.0
MOVL C04454 V=8.0
MOVL C04455 V=8.0
MOVL C04456 V=8.0
MOVL C04457 V=8.0
MOVL C04458 V=8.0
MOVL C04459 V=8.0
MOVL C04460 V=8.0
MOVL C04461 V=8.0
MOVL C04462 V=8.0
MOVL C04463 V=8.0
MOVL C04464 V=8.0
MOVJ C04465 VJ=0.78
MOVL C04466 V=8.0
MOVL C04467 V=8.0
MOVL C04468 V=8.0
MOVL C04469 V=8.0
MOVL C04470 V=8.0
MOVL C04471 V=8.0
MOVL C04472 V=8.0
MOVL C04473 V=8.0
MOVL C04474 V=8.0
MOVL C04475 V=8.0
MOVL C04476 V=8.0
MOVL C04477 V=8.0
MOVL C04478 V=8.0
MOVL C04479 V=8.0
MOVL C04480 V=8.0
MOVL C04481 V=8.0
MOVL C04482 V=8.0
MOVL C04483 V=8.0
MOVL C04484 V=8.0
MOVL C04485 V=8.0
MOVL C04486 V=8.0
MOVL C04487 V=8.0
MOVL C04488 V=8.0
MOVL C04489 V=8.0
MOVL C04490 V=8.0
MOVL C04491 V=8.0
MOVL C04492 V=8.0
MOVL C04493 V=8.0
MOVL C04494 V=8.0
MOVL C04495 V=8.0
MOVL C04496 V=8.0
MOVL C04497 V=8.0
MOVL C04498 V=8.0
MOVL C04499 V=8.0
MOVL C04500 V=8.0
MOVL C04501 V=8.0
MOVL C04502 V=8.0
MOVL C04503 V=8.0
MOVL C04504 V=8.0
MOVL C04505 V=8.0
MOVL C04506 V=8.0
MOVL C04507 V=8.0
MOVL C04508 V=8.0
MOVL C04509 V=8.0
MOVL C04510 V=8.0
MOVL C04511 V=8.0
MOVL C04512 V=8.0
MOVL C04513 V=8.0
MOVL C04514 V=8.0
MOVL C04515 V=8.0
MOVL C04516 V=8.0
MOVL C04517 V=8.0
MOVL C04518 V=8.0
MOVL C04519 V=8.0
MOVL C04520 V=8.0
MOVL C04521 V=8.0
MOVL C04522 V=8.0
MOVL C04523 V=8.0
MOVL C04524 V=8.0
MOVL C04525 V=8.0
MOVL C04526 V=8.0
MOVL C04527 V=8.0
MOVJ C04528 VJ=0.78
MOVL C04529 V=8.0
MOVL C04530 V=8.0
MOVL C04531 V=8.0
MOVL C04532 V=8.0
MOVL C04533 V=8.0
MOVL C04534 V=8.0
MOVL C04535 V=8.0
MOVL C04536 V=8.0
MOVL C04537 V=8.0
MOVL C04538 V=8.0
MOVL C04539 V=8.0
MOVL C04540 V=8.0
MOVL C04541 V=8.0
MOVL C04542 V=8.0
MOVL C04543 V=8.0
MOVL C04544 V=8.0
MOVL C04545 V=8.0
MOVL C04546 V=8.0
MOVL C04547 V=8.0
MOVL C04548 V=8.0
MOVL C04549 V=8.0
MOVJ C04550 VJ=0.78
MOVJ C04551 VJ=0.78
MOVL C04552 V=11.7
TIMER T=2.00
MOVL C04553 V=11.7
MOVJ C04554 VJ=0.78
MOVJ C04555 VJ=0.78
MOVL C04556 V=8.0
MOVL C04557 V=8.0
MOVL C04558 V=8.0
MOVL C04559 V=8.0
MOVL C04560 V=8.0
MOVL C04561 V=8.0
MOVL C04562 V=8.0
MOVL C04563 V=8.0
MOVL C04564 V=8.0
MOVL C04565 V=8.0
MOVL C04566 V=8.0
MOVL C04567 V=8.0
MOVL C04568 V=8.0
MOVL C04569 V=8.0
MOVL C04570 V=8.0
MOVL C04571 V=8.0
MOVL C04572 V=8.0
MOVL C04573 V=8.0
MOVL C04574 V=8.0
MOVL C04575 V=8.0
MOVL C04576 V=8.0
MOVL C04577 V=8.0
MOVL C04578 V=8.0
MOVL C04579 V=8.0
MOVL C04580 V=8.0
MOVL C04581 V=8.0
MOVL C04582 V=8.0
MOVL C04583 V=8.0
MOVL C04584 V=8.0
MOVL C04585 V=8.0
MOVL C04586 V=8.0
MOVL C04587 V=8.0
MOVL C04588 V=8.0
MOVL C04589 V=8.0
MOVL C04590 V=8.0
MOVL C04591 V=8.0
MOVL C04592 V=8.0
MOVL C04593 V=8.0
MOVL C04594 V=8.0
MOVL C04595 V=8.0
MOVL C04596 V=8.0
MOVL C04597 V=8.0
MOVJ C04598 VJ=0.78
MOVL C04599 V=8.0
MOVL C04600 V=8.0
MOVL C04601 V=8.0
MOVL C04602 V=8.0
MOVL C04603 V=8.0
MOVL C04604 V=8.0
MOVL C04605 V=8.0
MOVL C04606 V=8.0
MOVL C04607 V=8.0
MOVL C04608 V=8.0
MOVL C04609 V=8.0
MOVL C04610 V=8.0
MOVL C04611 V=8.0
MOVL C04612 V=8.0
MOVL C04613 V=8.0
MOVL C04614 V=8.0
MOVL C04615 V=8.0
MOVL C04616 V=8.0
MOVL C04617 V=8.0
MOVL C04618 V=8.0
MOVL C04619 V=8.0
MOVL C04620 V=8.0
MOVL C04621 V=8.0
MOVL C04622 V=8.0
MOVL C04623 V=8.0
MOVL C04624 V=8.0
MOVL C04625 V=8.0
MOVL C04626 V=8.0
MOVL C04627 V=8.0
MOVL C04628 V=8.0
MOVL C04629 V=8.0
MOVL C04630 V=8.0
MOVL C04631 V=8.0
MOVL C04632 V=8.0
MOVL C04633 V=8.0
MOVL C04634 V=8.0
MOVL C04635 V=8.0
MOVL C04636 V=8.0
MOVL C04637 V=8.0
MOVL C04638 V=8.0
MOVL C04639 V=8.0
MOVL C04640 V=8.0
MOVL C04641 V=8.0
MOVL C04642 V=8.0
MOVL C04643 V=8.0
MOVL C04644 V=8.0
MOVL C04645 V=8.0
MOVL C04646 V=8.0
MOVL C04647 V=8.0
MOVL C04648 V=8.0
MOVL C04649 V=8.0
MOVL C04650 V=8.0
MOVL C04651 V=8.0
MOVL C04652 V=8.0
MOVL C04653 V=8.0
MOVL C04654 V=8.0
MOVL C04655 V=8.0
MOVL C04656 V=8.0
MOVL C04657 V=8.0
MOVL C04658 V=8.0
MOVL C04659 V=8.0
MOVL C04660 V=8.0
MOVJ C04661 VJ=0.78
MOVL C04662 V=8.0
MOVL C04663 V=8.0
MOVL C04664 V=8.0
MOVL C04665 V=8.0
MOVL C04666 V=8.0
MOVL C04667 V=8.0
MOVL C04668 V=8.0
MOVL C04669 V=8.0
MOVL C04670 V=8.0
MOVL C04671 V=8.0
MOVL C04672 V=8.0
MOVL C04673 V=8.0
MOVL C04674 V=8.0
MOVL C04675 V=8.0
MOVL C04676 V=8.0
MOVL C04677 V=8.0
MOVL C04678 V=8.0
MOVL C04679 V=8.0
MOVL C04680 V=8.0
MOVL C04681 V=8.0
MOVL C04682 V=8.0
MOVL C04683 V=8.0
MOVL C04684 V=8.0
MOVL C04685 V=8.0
MOVL C04686 V=8.0
MOVL C04687 V=8.0
MOVL C04688 V=8.0
MOVL C04689 V=8.0
MOVL C04690 V=8.0
MOVL C04691 V=8.0
MOVL C04692 V=8.0
MOVL C04693 V=8.0
MOVL C04694 V=8.0
MOVL C04695 V=8.0
MOVL C04696 V=8.0
MOVL C04697 V=8.0
MOVL C04698 V=8.0
MOVL C04699 V=8.0
MOVL C04700 V=8.0
MOVL C04701 V=8.0
MOVL C04702 V=8.0
MOVL C04703 V=8.0
MOVL C04704 V=8.0
MOVL C04705 V=8.0
